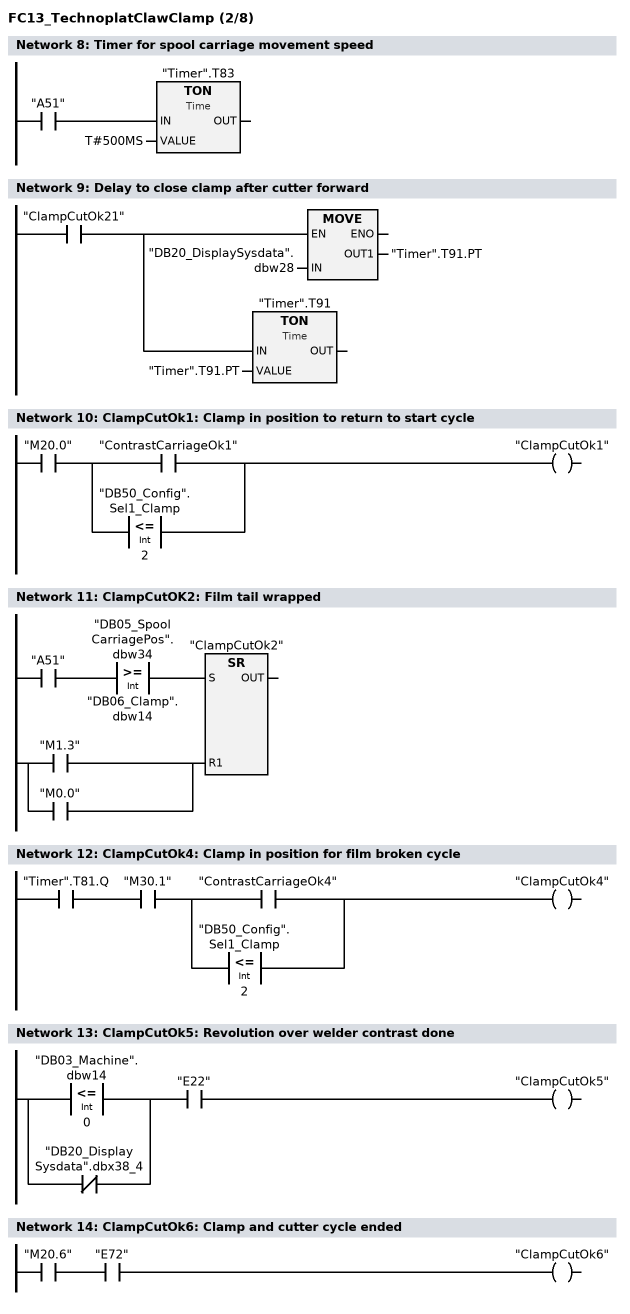
   "Timer".T83.TON(IN := "A51", PT := T#500MS);   // TON coil
END_REGION

REGION Network 9: Delay to close clamp after cutter forward
   IF "ClampCutOk21" THEN "Timer".T91.PT := "DB20_DisplaySysdata".dbw28; END_IF;
   "Timer".T91.TON(IN := "ClampCutOk21", PT := "Timer".T91.PT);   // TON coil
END_REGION

REGION Network 10: ClampCutOk1: Clamp in position to return to start cycle
   RUNG wire#powerrail
      Contact( "M20.0" )
      wire#w1
      Contact( "ContrastCarriageOk1" )
      wire#w2
      Coil( "ClampCutOk1" )
   END_RUNG
   RUNG wire#w1
      { S7_Templates := "SrcType := Int" } LE_Contact(in1 := "DB50_Config".Sel1_Clamp, in2 := 2)
   END_RUNG wire#w2
   // the same network as SCL:
   "ClampCutOk1" := "M20.0" AND ("ContrastCarriageOk1" OR ("DB50_Config".Sel1_Clamp <= 2));
END_REGION

REGION Network 11: ClampCutOK2: Film tail wrapped
   RUNG wire#powerrail
      Contact( "A51" )
      { S7_Templates := "SrcType := Int" } GE_Contact(in1 := "DB05_SpoolCarriagePos".dbw34, in2 := "DB06_Clamp".dbw14)
      S_SR(operand := "ClampCutOk2", r1 := wire#w1)
   END_RUNG
   RUNG wire#powerrail
      Contact( "M1.3" )
   END_RUNG wire#w1
   RUNG wire#powerrail
      Contact( "M0.0" )
   END_RUNG wire#w1
   // the same network as SCL:
   IF "A51" AND ("DB05_SpoolCarriagePos".dbw34 >= "DB06_Clamp".dbw14) THEN
       "ClampCutOk2" := TRUE;   // SR flip-flop
   END_IF;
   IF "M1.3" OR "M0.0" THEN "ClampCutOk2" := FALSE; END_IF;
END_REGION

REGION Network 12: ClampCutOk4: Clamp in position for film broken cycle
   RUNG wire#powerrail
      Contact( "Timer".T81.Q )
      Contact( "M30.1" )
      wire#w1
      Contact( "ContrastCarriageOk4" )
      wire#w2
      Coil( "ClampCutOk4" )
   END_RUNG
   RUNG wire#w1
      { S7_Templates := "SrcType := Int" } LE_Contact(in1 := "DB50_Config".Sel1_Clamp, in2 := 2)
   END_RUNG wire#w2
   // the same network as SCL:
   "ClampCutOk4" := "Timer".T81.Q AND "M30.1" AND ("ContrastCarriageOk4" OR ("DB50_Config".Sel1_Clamp <= 2));
END_REGION

REGION Network 13: ClampCutOk5: Revolution over welder contrast done
   RUNG wire#powerrail
      { S7_Templates := "SrcType := Int" } LE_Contact(in1 := "DB03_Machine".dbw14, in2 := 0)
      wire#w1
      Contact( "E22" )
      Coil( "ClampCutOk5" )
   END_RUNG
   RUNG wire#powerrail
      I_Contact( "DB20_DisplaySysdata".dbx38_4 )
   END_RUNG wire#w1
   // the same network as SCL:
   "ClampCutOk5" := (("DB03_Machine".dbw14 <= 0) OR NOT "DB20_DisplaySysdata".dbx38_4) AND "E22";
END_REGION

REGION Network 14: ClampCutOk6: Clamp and cutter cycle ended
   RUNG wire#powerrail
      Contact( "M20.6" )
      Contact( "E72" )
      Coil( "ClampCutOk6" )
   END_RUNG
   // the same network as SCL:
   "ClampCutOk6" := "M20.6" AND "E72";
END_REGION

REGION Network 15: ClampCutOk7: Clamp and cutter units in position to begin cycle
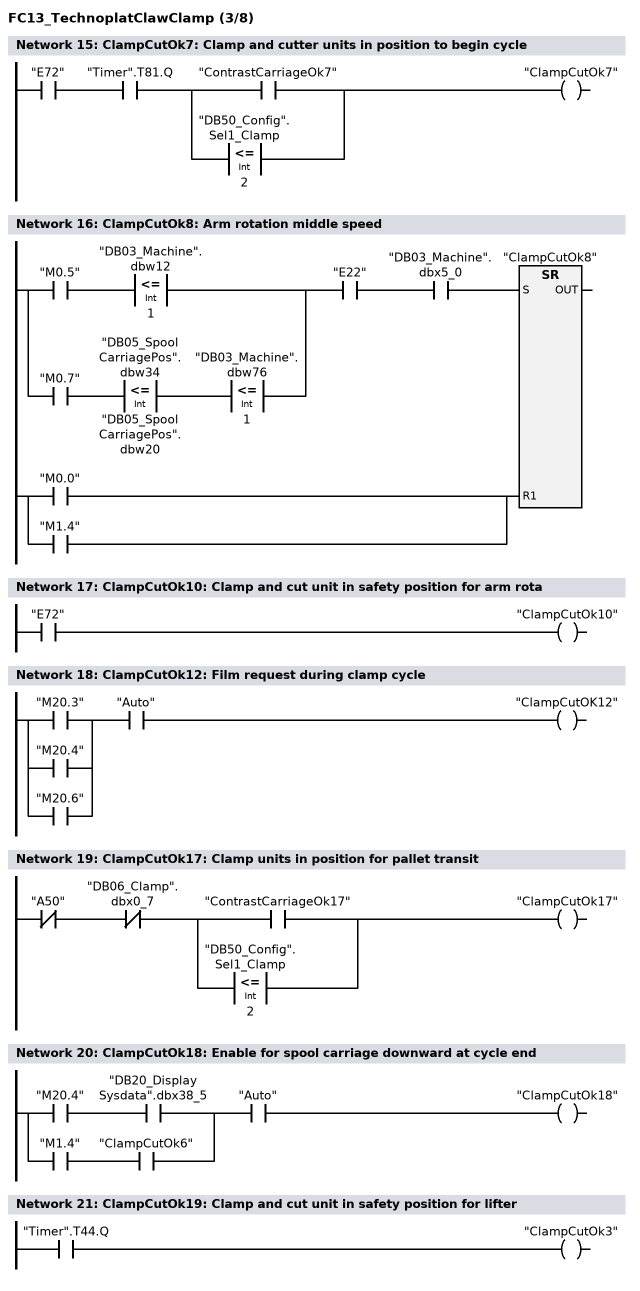
   RUNG wire#powerrail
      Contact( "E72" )
      Contact( "Timer".T81.Q )
      wire#w1
      Contact( "ContrastCarriageOk7" )
      wire#w2
      Coil( "ClampCutOk7" )
   END_RUNG
   RUNG wire#w1
      { S7_Templates := "SrcType := Int" } LE_Contact(in1 := "DB50_Config".Sel1_Clamp, in2 := 2)
   END_RUNG wire#w2
   // the same network as SCL:
   "ClampCutOk7" := "E72" AND "Timer".T81.Q AND ("ContrastCarriageOk7" OR ("DB50_Config".Sel1_Clamp <= 2));
END_REGION

REGION Network 16: ClampCutOk8: Arm rotation middle speed
   RUNG wire#powerrail
      Contact( "M0.5" )
      { S7_Templates := "SrcType := Int" } LE_Contact(in1 := "DB03_Machine".dbw12, in2 := 1)
      wire#w1
      Contact( "E22" )
      Contact( "DB03_Machine".dbx5_0 )
      S_SR(operand := "ClampCutOk8", r1 := wire#w2)
   END_RUNG
   RUNG wire#powerrail
      Contact( "M0.7" )
      { S7_Templates := "SrcType := Int" } LE_Contact(in1 := "DB05_SpoolCarriagePos".dbw34, in2 := "DB05_SpoolCarriagePos".dbw20)
      { S7_Templates := "SrcType := Int" } LE_Contact(in1 := "DB03_Machine".dbw76, in2 := 1)
   END_RUNG wire#w1
   RUNG wire#powerrail
      Contact( "M0.0" )
   END_RUNG wire#w2
   RUNG wire#powerrail
      Contact( "M1.4" )
   END_RUNG wire#w2
   // the same network as SCL:
   IF (("M0.5" AND ("DB03_Machine".dbw12 <= 1)) OR ("M0.7" AND ("DB05_SpoolCarriagePos".dbw34 <= "DB05_SpoolCarriagePos".dbw20) AND ("DB03_Machine".dbw76 <= 1))) AND "E22" AND "DB03_Machine".dbx5_0 THEN
       "ClampCutOk8" := TRUE;   // SR flip-flop
   END_IF;
   IF "M0.0" OR "M1.4" THEN "ClampCutOk8" := FALSE; END_IF;
END_REGION

REGION Network 17: ClampCutOk10: Clamp and cut unit in safety position for arm rota
   RUNG wire#powerrail
      Contact( "E72" )
      Coil( "ClampCutOk10" )
   END_RUNG
   // the same network as SCL:
   "ClampCutOk10" := "E72";
END_REGION

REGION Network 18: ClampCutOk12: Film request during clamp cycle
   RUNG wire#powerrail
      Contact( "M20.3" )
      wire#w1
      Contact( "Auto" )
      Coil( "ClampCutOK12" )
   END_RUNG
   RUNG wire#powerrail
      Contact( "M20.4" )
   END_RUNG wire#w1
   RUNG wire#powerrail
      Contact( "M20.6" )
   END_RUNG wire#w1
   // the same network as SCL:
   "ClampCutOK12" := ("M20.3" OR "M20.4" OR "M20.6") AND "Auto";
END_REGION

REGION Network 19: ClampCutOk17: Clamp units in position for pallet transit
   RUNG wire#powerrail
      I_Contact( "A50" )
      I_Contact( "DB06_Clamp".dbx0_7 )
      wire#w1
      Contact( "ContrastCarriageOk17" )
      wire#w2
      Coil( "ClampCutOk17" )
   END_RUNG
   RUNG wire#w1
      { S7_Templates := "SrcType := Int" } LE_Contact(in1 := "DB50_Config".Sel1_Clamp, in2 := 2)
   END_RUNG wire#w2
   // the same network as SCL:
   "ClampCutOk17" := NOT "A50" AND NOT "DB06_Clamp".dbx0_7 AND ("ContrastCarriageOk17" OR ("DB50_Config".Sel1_Clamp <= 2));
END_REGION

REGION Network 20: ClampCutOk18: Enable for spool carriage downward at cycle end
   RUNG wire#powerrail
      Contact( "M20.4" )
      Contact( "DB20_DisplaySysdata".dbx38_5 )
      wire#w1
      Contact( "Auto" )
      Coil( "ClampCutOk18" )
   END_RUNG
   RUNG wire#powerrail
      Contact( "M1.4" )
      Contact( "ClampCutOk6" )
   END_RUNG wire#w1
   // the same network as SCL:
   "ClampCutOk18" := (("M20.4" AND "DB20_DisplaySysdata".dbx38_5) OR ("M1.4" AND "ClampCutOk6")) AND "Auto";
END_REGION

REGION Network 21: ClampCutOk19: Clamp and cut unit in safety position for lifter
   RUNG wire#powerrail
      Contact( "Timer".T44.Q )
      Coil( "ClampCutOk3" )
   END_RUNG
   // the same network as SCL:
   "ClampCutOk3" := "Timer".T44.Q;
END_REGION

REGION Network 22: ClampCutOk11: Exclude deceleration not correct alarm
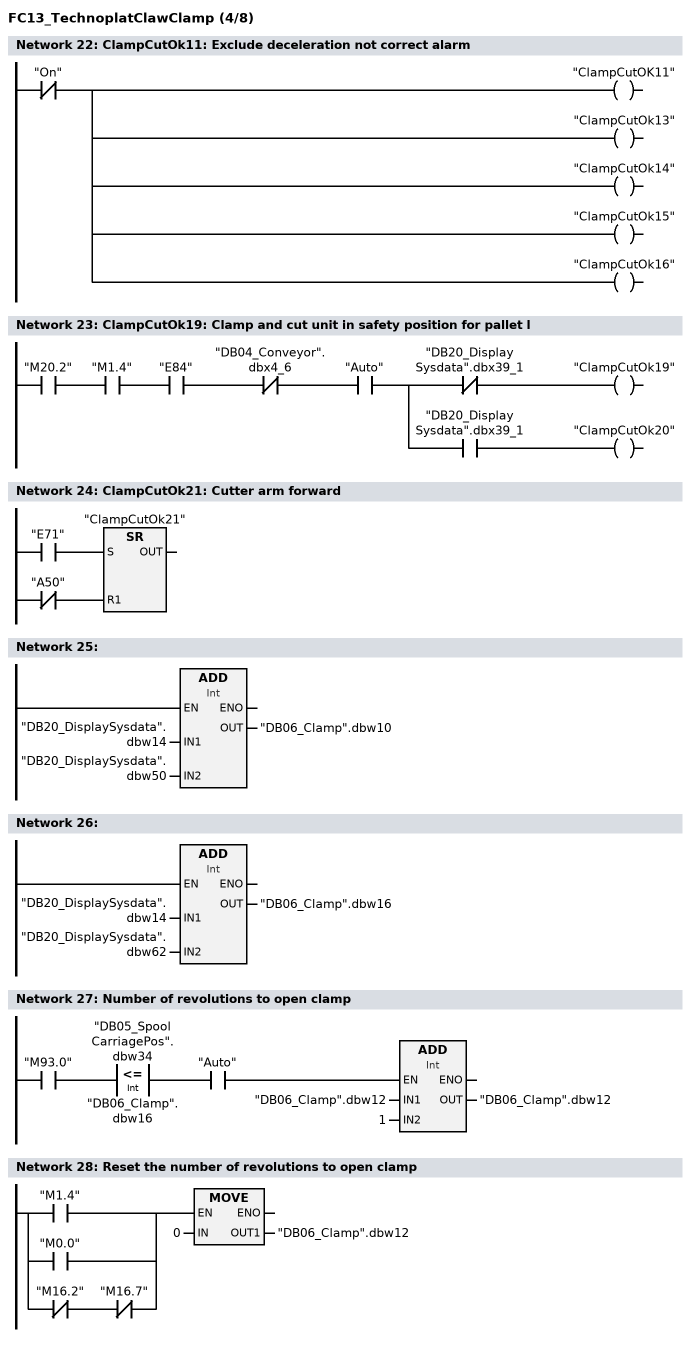
   RUNG wire#powerrail
      I_Contact( "On" )
      wire#w1
      Coil( "ClampCutOK11" )
   END_RUNG
   RUNG wire#w1
      Coil( "ClampCutOk13" )
   END_RUNG
   RUNG wire#w1
      Coil( "ClampCutOk14" )
   END_RUNG
   RUNG wire#w1
      Coil( "ClampCutOk15" )
   END_RUNG
   RUNG wire#w1
      Coil( "ClampCutOk16" )
   END_RUNG
   // the same network as SCL:
   "ClampCutOK11" := NOT "On";
   "ClampCutOk13" := NOT "On";
   "ClampCutOk14" := NOT "On";
   "ClampCutOk15" := NOT "On";
   "ClampCutOk16" := NOT "On";
END_REGION

REGION Network 23: ClampCutOk19: Clamp and cut unit in safety position for pallet l
   RUNG wire#powerrail
      Contact( "M20.2" )
      Contact( "M1.4" )
      Contact( "E84" )
      I_Contact( "DB04_Conveyor".dbx4_6 )
      Contact( "Auto" )
      wire#w1
      I_Contact( "DB20_DisplaySysdata".dbx39_1 )
      Coil( "ClampCutOk19" )
   END_RUNG
   RUNG wire#w1
      Contact( "DB20_DisplaySysdata".dbx39_1 )
      Coil( "ClampCutOk20" )
   END_RUNG
   // the same network as SCL:
   #_w1 := "M20.2" AND "M1.4" AND "E84" AND NOT "DB04_Conveyor".dbx4_6 AND "Auto";
   "ClampCutOk19" := #_w1 AND NOT "DB20_DisplaySysdata".dbx39_1;
   "ClampCutOk20" := #_w1 AND "DB20_DisplaySysdata".dbx39_1;
END_REGION

REGION Network 24: ClampCutOk21: Cutter arm forward
   RUNG wire#powerrail
      Contact( "E71" )
      S_SR(operand := "ClampCutOk21", r1 := wire#w1)
   END_RUNG
   RUNG wire#powerrail
      I_Contact( "A50" )
   END_RUNG wire#w1
   // the same network as SCL:
   IF "E71" THEN
       "ClampCutOk21" := TRUE;   // SR flip-flop
   END_IF;
   IF NOT "A50" THEN "ClampCutOk21" := FALSE; END_IF;
END_REGION

REGION Network 25
   RUNG wire#powerrail
      { S7_Templates := "SrcType := Int"; S7_GenerateENO := "TRUE" } Add(in1 := "DB20_DisplaySysdata".dbw14, in2 := "DB20_DisplaySysdata".dbw50, out => "DB06_Clamp".dbw10)
   END_RUNG
   // the same network as SCL:
   "DB06_Clamp".dbw10 := "DB20_DisplaySysdata".dbw14 + "DB20_DisplaySysdata".dbw50;
END_REGION

REGION Network 26
   RUNG wire#powerrail
      { S7_Templates := "SrcType := Int"; S7_GenerateENO := "TRUE" } Add(in1 := "DB20_DisplaySysdata".dbw14, in2 := "DB20_DisplaySysdata".dbw62, out => "DB06_Clamp".dbw16)
   END_RUNG
   // the same network as SCL:
   "DB06_Clamp".dbw16 := "DB20_DisplaySysdata".dbw14 + "DB20_DisplaySysdata".dbw62;
END_REGION

REGION Network 27: Number of revolutions to open clamp
   RUNG wire#powerrail
      Contact( "M93.0" )
      { S7_Templates := "SrcType := Int" } LE_Contact(in1 := "DB05_SpoolCarriagePos".dbw34, in2 := "DB06_Clamp".dbw16)
      Contact( "Auto" )
      { S7_Templates := "SrcType := Int"; S7_GenerateENO := "TRUE" } Add(in1 := "DB06_Clamp".dbw12, in2 := 1, out => "DB06_Clamp".dbw12)
   END_RUNG
   // the same network as SCL:
   IF "M93.0" AND ("DB05_SpoolCarriagePos".dbw34 <= "DB06_Clamp".dbw16) AND "Auto" THEN
       "DB06_Clamp".dbw12 := "DB06_Clamp".dbw12 + 1;
   END_IF;
END_REGION

REGION Network 28: Reset the number of revolutions to open clamp
   RUNG wire#powerrail
      Contact( "M1.4" )
      wire#w1
      { S7_GenerateENO := "TRUE" } Move(in := 0, out1 => "DB06_Clamp".dbw12)
   END_RUNG
   RUNG wire#powerrail
      Contact( "M0.0" )
   END_RUNG wire#w1
   RUNG wire#powerrail
      I_Contact( "M16.2" )
      I_Contact( "M16.7" )
   END_RUNG wire#w1
   // the same network as SCL:
   IF "M1.4" OR "M0.0" OR (NOT "M16.2" AND NOT "M16.7") THEN "DB06_Clamp".dbw12 := 0; END_IF;
END_REGION

REGION Network 29
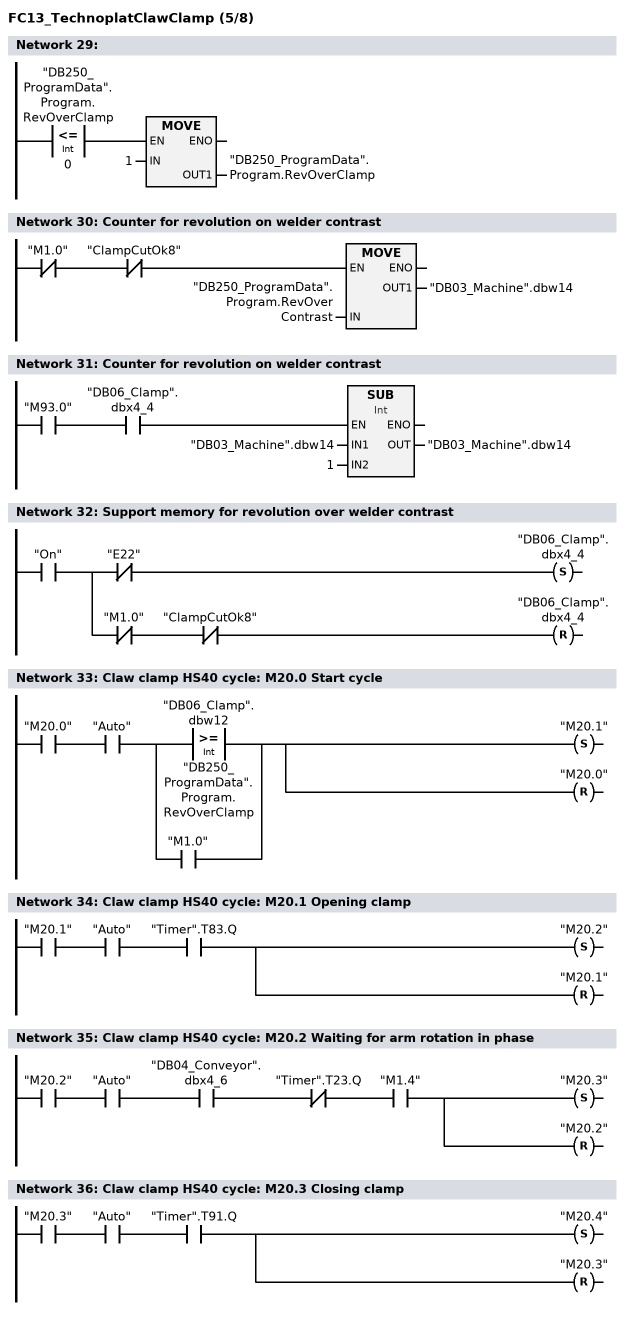
   RUNG wire#powerrail
      { S7_Templates := "SrcType := Int" } LE_Contact(in1 := "DB250_ProgramData".Program.RevOverClamp, in2 := 0)
      { S7_GenerateENO := "TRUE" } Move(in := 1, out1 => "DB250_ProgramData".Program.RevOverClamp)
   END_RUNG
   // the same network as SCL:
   IF "DB250_ProgramData".Program.RevOverClamp <= 0 THEN
       "DB250_ProgramData".Program.RevOverClamp := 1;
   END_IF;
END_REGION

REGION Network 30: Counter for revolution on welder contrast
   RUNG wire#powerrail
      I_Contact( "M1.0" )
      I_Contact( "ClampCutOk8" )
      { S7_GenerateENO := "TRUE" } Move(in := "DB250_ProgramData".Program.RevOverContrast, out1 => "DB03_Machine".dbw14)
   END_RUNG
   // the same network as SCL:
   IF NOT "M1.0" AND NOT "ClampCutOk8" THEN
       "DB03_Machine".dbw14 := "DB250_ProgramData".Program.RevOverContrast;
   END_IF;
END_REGION

REGION Network 31: Counter for revolution on welder contrast
   RUNG wire#powerrail
      Contact( "M93.0" )
      Contact( "DB06_Clamp".dbx4_4 )
      { S7_Templates := "SrcType := Int"; S7_GenerateENO := "TRUE" } Sub(in1 := "DB03_Machine".dbw14, in2 := 1, out => "DB03_Machine".dbw14)
   END_RUNG
   // the same network as SCL:
   IF "M93.0" AND "DB06_Clamp".dbx4_4 THEN "DB03_Machine".dbw14 := "DB03_Machine".dbw14 - 1; END_IF;
END_REGION

REGION Network 32: Support memory for revolution over welder contrast
   RUNG wire#powerrail
      Contact( "On" )
      wire#w1
      I_Contact( "E22" )
      S_Coil( "DB06_Clamp".dbx4_4 )
   END_RUNG
   RUNG wire#w1
      I_Contact( "M1.0" )
      I_Contact( "ClampCutOk8" )
      R_Coil( "DB06_Clamp".dbx4_4 )
   END_RUNG
   // the same network as SCL:
   IF "On" AND NOT "E22" THEN "DB06_Clamp".dbx4_4 := TRUE; END_IF;
   IF "On" AND NOT "M1.0" AND NOT "ClampCutOk8" THEN "DB06_Clamp".dbx4_4 := FALSE; END_IF;
END_REGION

REGION Network 33: Claw clamp HS40 cycle: M20.0 Start cycle
   RUNG wire#powerrail
      Contact( "M20.0" )
      Contact( "Auto" )
      wire#w1
      { S7_Templates := "SrcType := Int" } GE_Contact(in1 := "DB06_Clamp".dbw12, in2 := "DB250_ProgramData".Program.RevOverClamp)
      wire#w2
      S_Coil( "M20.1" )
   END_RUNG
   RUNG wire#w1
      Contact( "M1.0" )
   END_RUNG wire#w2
   RUNG wire#w2
      R_Coil( "M20.0" )
   END_RUNG
   // the same network as SCL:
   IF "M20.0" AND "Auto" AND (("DB06_Clamp".dbw12 >= "DB250_ProgramData".Program.RevOverClamp) OR "M1.0") THEN
       "M20.1" := TRUE;
       "M20.0" := FALSE;
   END_IF;
END_REGION

REGION Network 34: Claw clamp HS40 cycle: M20.1 Opening clamp
   RUNG wire#powerrail
      Contact( "M20.1" )
      Contact( "Auto" )
      Contact( "Timer".T83.Q )
      wire#w1
      S_Coil( "M20.2" )
   END_RUNG
   RUNG wire#w1
      R_Coil( "M20.1" )
   END_RUNG
   // the same network as SCL:
   IF "M20.1" AND "Auto" AND "Timer".T83.Q THEN
       "M20.2" := TRUE;
       "M20.1" := FALSE;
   END_IF;
END_REGION

REGION Network 35: Claw clamp HS40 cycle: M20.2 Waiting for arm rotation in phase
   RUNG wire#powerrail
      Contact( "M20.2" )
      Contact( "Auto" )
      Contact( "DB04_Conveyor".dbx4_6 )
      I_Contact( "Timer".T23.Q )
      Contact( "M1.4" )
      wire#w1
      S_Coil( "M20.3" )
   END_RUNG
   RUNG wire#w1
      R_Coil( "M20.2" )
   END_RUNG
   // the same network as SCL:
   IF "M20.2" AND "Auto" AND "DB04_Conveyor".dbx4_6 AND NOT "Timer".T23.Q AND "M1.4" THEN
       "M20.3" := TRUE;
       "M20.2" := FALSE;
   END_IF;
END_REGION

REGION Network 36: Claw clamp HS40 cycle: M20.3 Closing clamp
   RUNG wire#powerrail
      Contact( "M20.3" )
      Contact( "Auto" )
      Contact( "Timer".T91.Q )
      wire#w1
      S_Coil( "M20.4" )
   END_RUNG
   RUNG wire#w1
      R_Coil( "M20.3" )
   END_RUNG
   // the same network as SCL:
   IF "M20.3" AND "Auto" AND "Timer".T91.Q THEN
       "M20.4" := TRUE;
       "M20.3" := FALSE;
   END_IF;
END_REGION

REGION Network 37: Claw clamp HS40 cycle: M20.4 Welder and cut unit forward
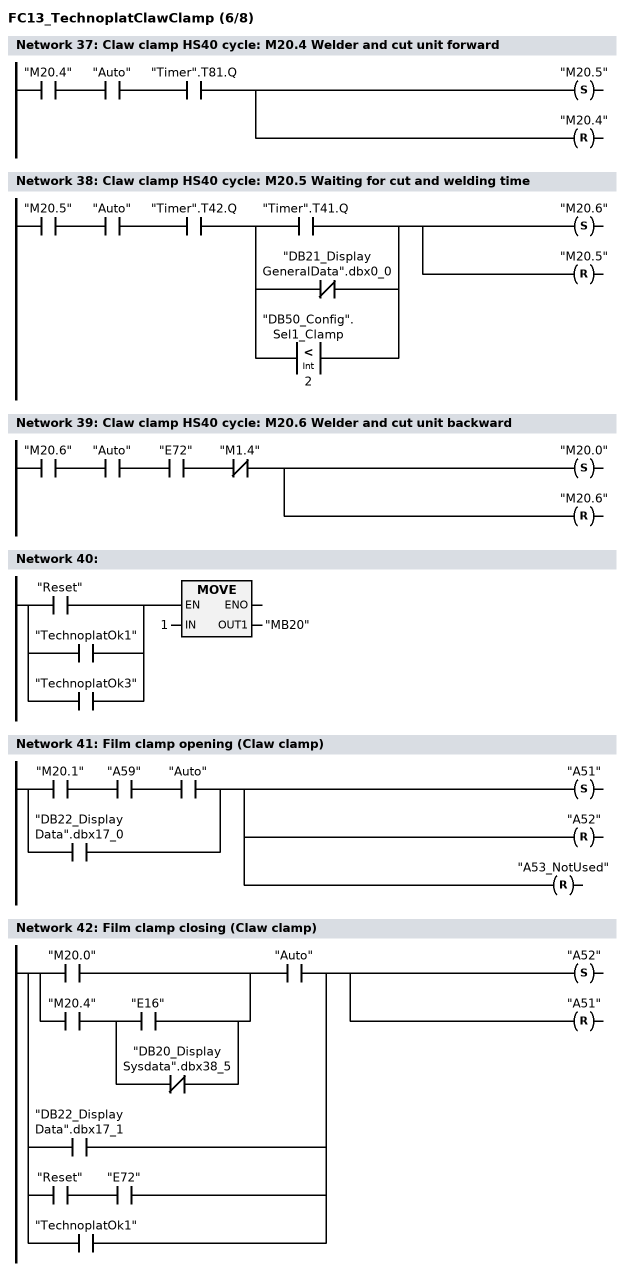
   RUNG wire#powerrail
      Contact( "M20.4" )
      Contact( "Auto" )
      Contact( "Timer".T81.Q )
      wire#w1
      S_Coil( "M20.5" )
   END_RUNG
   RUNG wire#w1
      R_Coil( "M20.4" )
   END_RUNG
   // the same network as SCL:
   IF "M20.4" AND "Auto" AND "Timer".T81.Q THEN
       "M20.5" := TRUE;
       "M20.4" := FALSE;
   END_IF;
END_REGION

REGION Network 38: Claw clamp HS40 cycle: M20.5 Waiting for cut and welding time
   RUNG wire#powerrail
      Contact( "M20.5" )
      Contact( "Auto" )
      Contact( "Timer".T42.Q )
      wire#w1
      Contact( "Timer".T41.Q )
      wire#w2
      S_Coil( "M20.6" )
   END_RUNG
   RUNG wire#w1
      I_Contact( "DB21_DisplayGeneralData".dbx0_0 )
   END_RUNG wire#w2
   RUNG wire#w1
      { S7_Templates := "SrcType := Int" } LT_Contact(in1 := "DB50_Config".Sel1_Clamp, in2 := 2)
   END_RUNG wire#w2
   RUNG wire#w2
      R_Coil( "M20.5" )
   END_RUNG
   // the same network as SCL:
   IF "M20.5" AND "Auto" AND "Timer".T42.Q AND ("Timer".T41.Q OR NOT "DB21_DisplayGeneralData".dbx0_0 OR ("DB50_Config".Sel1_Clamp < 2)) THEN
       "M20.6" := TRUE;
       "M20.5" := FALSE;
   END_IF;
END_REGION

REGION Network 39: Claw clamp HS40 cycle: M20.6 Welder and cut unit backward
   RUNG wire#powerrail
      Contact( "M20.6" )
      Contact( "Auto" )
      Contact( "E72" )
      I_Contact( "M1.4" )
      wire#w1
      S_Coil( "M20.0" )
   END_RUNG
   RUNG wire#w1
      R_Coil( "M20.6" )
   END_RUNG
   // the same network as SCL:
   IF "M20.6" AND "Auto" AND "E72" AND NOT "M1.4" THEN
       "M20.0" := TRUE;
       "M20.6" := FALSE;
   END_IF;
END_REGION

REGION Network 40
   RUNG wire#powerrail
      Contact( "Reset" )
      wire#w1
      { S7_GenerateENO := "TRUE" } Move(in := 1, out1 => "MB20")
   END_RUNG
   RUNG wire#powerrail
      Contact( "TechnoplatOk1" )
   END_RUNG wire#w1
   RUNG wire#powerrail
      Contact( "TechnoplatOk3" )
   END_RUNG wire#w1
   // the same network as SCL:
   IF "Reset" OR "TechnoplatOk1" OR "TechnoplatOk3" THEN "MB20" := 1; END_IF;
END_REGION

REGION Network 41: Film clamp opening (Claw clamp)
   RUNG wire#powerrail
      Contact( "M20.1" )
      Contact( "A59" )
      Contact( "Auto" )
      wire#w1
      S_Coil( "A51" )
   END_RUNG
   RUNG wire#powerrail
      Contact( "DB22_DisplayData".dbx17_0 )
   END_RUNG wire#w1
   RUNG wire#w1
      R_Coil( "A52" )
   END_RUNG
   RUNG wire#w1
      R_Coil( "A53_NotUsed" )
   END_RUNG
   // the same network as SCL:
   IF ("M20.1" AND "A59" AND "Auto") OR "DB22_DisplayData".dbx17_0 THEN
       "A51" := TRUE;
       "A52" := FALSE;
       "A53_NotUsed" := FALSE;
   END_IF;
END_REGION

REGION Network 42: Film clamp closing (Claw clamp)
   RUNG wire#powerrail
      Contact( "M20.0" )
      wire#w1
      Contact( "Auto" )
      wire#w3
      S_Coil( "A52" )
   END_RUNG
   RUNG wire#powerrail
      Contact( "M20.4" )
      wire#w2
      Contact( "E16" )
   END_RUNG wire#w1
   RUNG wire#w2
      I_Contact( "DB20_DisplaySysdata".dbx38_5 )
   END_RUNG wire#w1
   RUNG wire#powerrail
      Contact( "DB22_DisplayData".dbx17_1 )
   END_RUNG wire#w3
   RUNG wire#powerrail
      Contact( "Reset" )
      Contact( "E72" )
   END_RUNG wire#w3
   RUNG wire#powerrail
      Contact( "TechnoplatOk1" )
   END_RUNG wire#w3
   RUNG wire#w3
      R_Coil( "A51" )
   END_RUNG
   // the same network as SCL:
   IF (("M20.0" OR ("M20.4" AND ("E16" OR NOT "DB20_DisplaySysdata".dbx38_5))) AND "Auto") OR "DB22_DisplayData".dbx17_1 OR ("Reset" AND "E72") OR "TechnoplatOk1" THEN
       "A52" := TRUE;
       "A51" := FALSE;
   END_IF;
END_REGION

REGION Network 43: Film clamp double closing (Claw clamp)
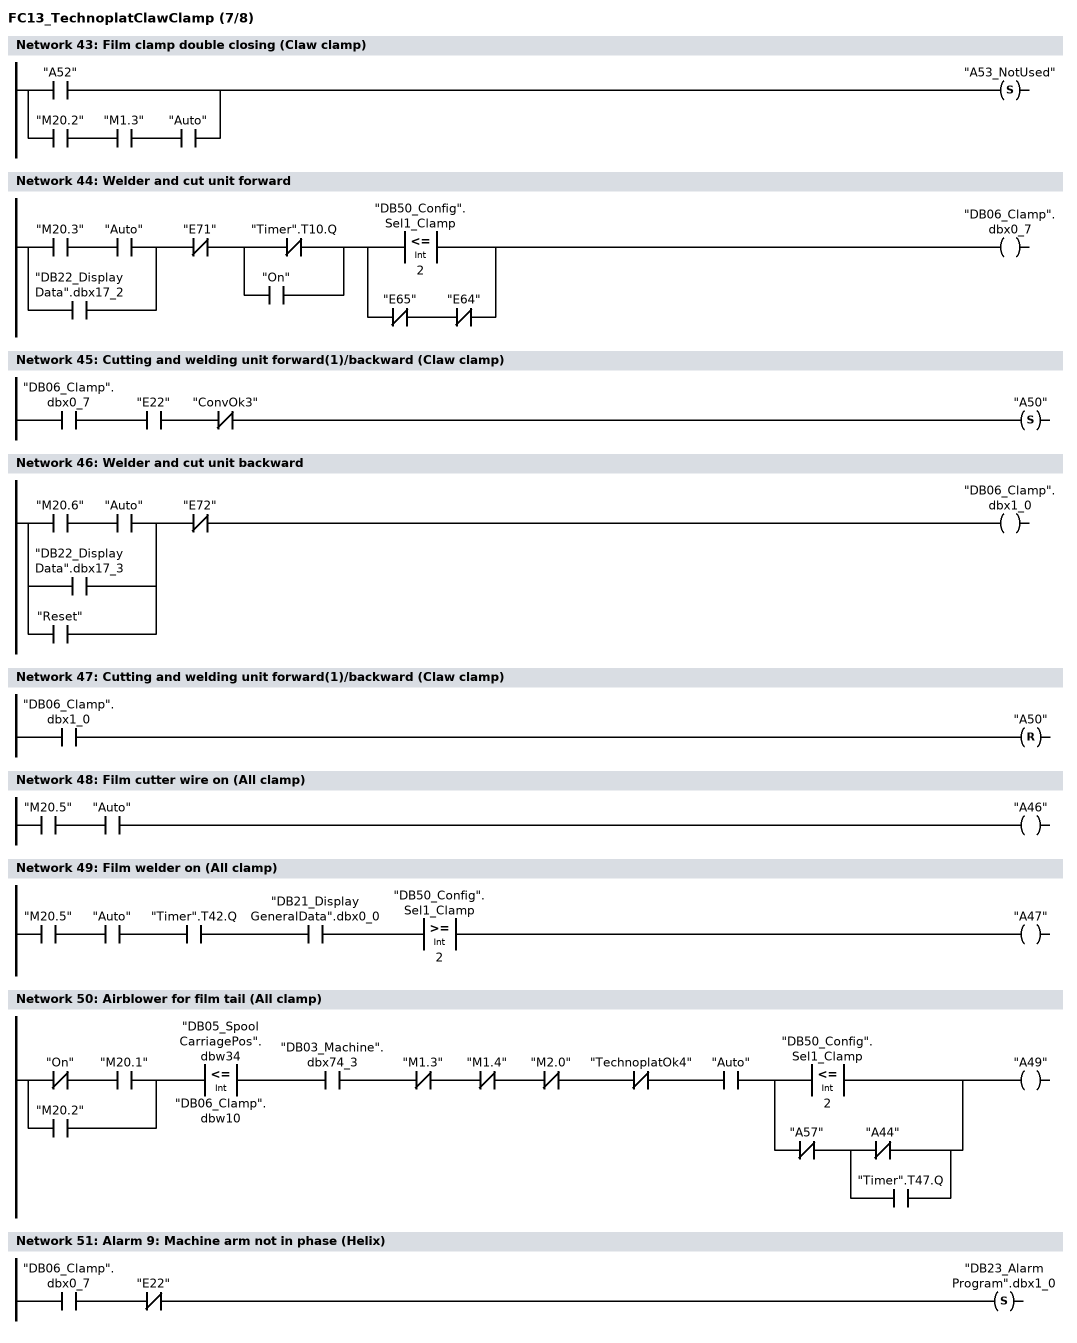
   RUNG wire#powerrail
      Contact( "A52" )
      wire#w1
      S_Coil( "A53_NotUsed" )
   END_RUNG
   RUNG wire#powerrail
      Contact( "M20.2" )
      Contact( "M1.3" )
      Contact( "Auto" )
   END_RUNG wire#w1
   // the same network as SCL:
   IF "A52" OR ("M20.2" AND "M1.3" AND "Auto") THEN "A53_NotUsed" := TRUE; END_IF;
END_REGION

REGION Network 44: Welder and cut unit forward
   RUNG wire#powerrail
      Contact( "M20.3" )
      Contact( "Auto" )
      wire#w1
      I_Contact( "E71" )
      wire#w2
      I_Contact( "Timer".T10.Q )
      wire#w3
      { S7_Templates := "SrcType := Int" } LE_Contact(in1 := "DB50_Config".Sel1_Clamp, in2 := 2)
      wire#w4
      Coil( "DB06_Clamp".dbx0_7 )
   END_RUNG
   RUNG wire#powerrail
      Contact( "DB22_DisplayData".dbx17_2 )
   END_RUNG wire#w1
   RUNG wire#w2
      Contact( "On" )
   END_RUNG wire#w3
   RUNG wire#w3
      I_Contact( "E65" )
      I_Contact( "E64" )
   END_RUNG wire#w4
   // the same network as SCL:
   "DB06_Clamp".dbx0_7 := (("M20.3" AND "Auto") OR "DB22_DisplayData".dbx17_2) AND NOT "E71" AND (NOT "Timer".T10.Q OR "On") AND (("DB50_Config".Sel1_Clamp <= 2) OR (NOT "E65" AND NOT "E64"));
END_REGION

REGION Network 45: Cutting and welding unit forward(1)/backward (Claw clamp)
   RUNG wire#powerrail
      Contact( "DB06_Clamp".dbx0_7 )
      Contact( "E22" )
      I_Contact( "ConvOk3" )
      S_Coil( "A50" )
   END_RUNG
   // the same network as SCL:
   IF "DB06_Clamp".dbx0_7 AND "E22" AND NOT "ConvOk3" THEN "A50" := TRUE; END_IF;
END_REGION

REGION Network 46: Welder and cut unit backward
   RUNG wire#powerrail
      Contact( "M20.6" )
      Contact( "Auto" )
      wire#w1
      I_Contact( "E72" )
      Coil( "DB06_Clamp".dbx1_0 )
   END_RUNG
   RUNG wire#powerrail
      Contact( "DB22_DisplayData".dbx17_3 )
   END_RUNG wire#w1
   RUNG wire#powerrail
      Contact( "Reset" )
   END_RUNG wire#w1
   // the same network as SCL:
   "DB06_Clamp".dbx1_0 := (("M20.6" AND "Auto") OR "DB22_DisplayData".dbx17_3 OR "Reset") AND NOT "E72";
END_REGION

REGION Network 47: Cutting and welding unit forward(1)/backward (Claw clamp)
   RUNG wire#powerrail
      Contact( "DB06_Clamp".dbx1_0 )
      R_Coil( "A50" )
   END_RUNG
   // the same network as SCL:
   IF "DB06_Clamp".dbx1_0 THEN "A50" := FALSE; END_IF;
END_REGION

REGION Network 48: Film cutter wire on (All clamp)
   RUNG wire#powerrail
      Contact( "M20.5" )
      Contact( "Auto" )
      Coil( "A46" )
   END_RUNG
   // the same network as SCL:
   "A46" := "M20.5" AND "Auto";
END_REGION

REGION Network 49: Film welder on (All clamp)
   RUNG wire#powerrail
      Contact( "M20.5" )
      Contact( "Auto" )
      Contact( "Timer".T42.Q )
      Contact( "DB21_DisplayGeneralData".dbx0_0 )
      { S7_Templates := "SrcType := Int" } GE_Contact(in1 := "DB50_Config".Sel1_Clamp, in2 := 2)
      Coil( "A47" )
   END_RUNG
   // the same network as SCL:
   "A47" := "M20.5" AND "Auto" AND "Timer".T42.Q AND "DB21_DisplayGeneralData".dbx0_0 AND ("DB50_Config".Sel1_Clamp >= 2);
END_REGION

REGION Network 50: Airblower for film tail (All clamp)
   RUNG wire#powerrail
      I_Contact( "On" )
      Contact( "M20.1" )
      wire#w1
      { S7_Templates := "SrcType := Int" } LE_Contact(in1 := "DB05_SpoolCarriagePos".dbw34, in2 := "DB06_Clamp".dbw10)
      Contact( "DB03_Machine".dbx74_3 )
      I_Contact( "M1.3" )
      I_Contact( "M1.4" )
      I_Contact( "M2.0" )
      I_Contact( "TechnoplatOk4" )
      Contact( "Auto" )
      wire#w2
      { S7_Templates := "SrcType := Int" } LE_Contact(in1 := "DB50_Config".Sel1_Clamp, in2 := 2)
      wire#w3
      Coil( "A49" )
   END_RUNG
   RUNG wire#powerrail
      Contact( "M20.2" )
   END_RUNG wire#w1
   RUNG wire#w2
      I_Contact( "A57" )
      wire#w4
      I_Contact( "A44" )
   END_RUNG wire#w3
   RUNG wire#w4
      Contact( "Timer".T47.Q )
   END_RUNG wire#w3
   // the same network as SCL:
   "A49" := ((NOT "On" AND "M20.1") OR "M20.2") AND ("DB05_SpoolCarriagePos".dbw34 <= "DB06_Clamp".dbw10) AND "DB03_Machine".dbx74_3 AND NOT "M1.3" AND NOT "M1.4" AND NOT "M2.0" AND NOT "TechnoplatOk4" AND "Auto" AND (("DB50_Config".Sel1_Clamp <= 2) OR (NOT "A57" AND (NOT "A44" OR "Timer".T47.Q)));
END_REGION

REGION Network 51: Alarm 9: Machine arm not in phase (Helix)
   RUNG wire#powerrail
      Contact( "DB06_Clamp".dbx0_7 )
      I_Contact( "E22" )
      S_Coil( "DB23_AlarmProgram".dbx1_0 )
   END_RUNG
   // the same network as SCL:
   IF "DB06_Clamp".dbx0_7 AND NOT "E22" THEN "DB23_AlarmProgram".dbx1_0 := TRUE; END_IF;
END_REGION

REGION Network 52: Alarm 52: Check the welder circuit (Clamp)
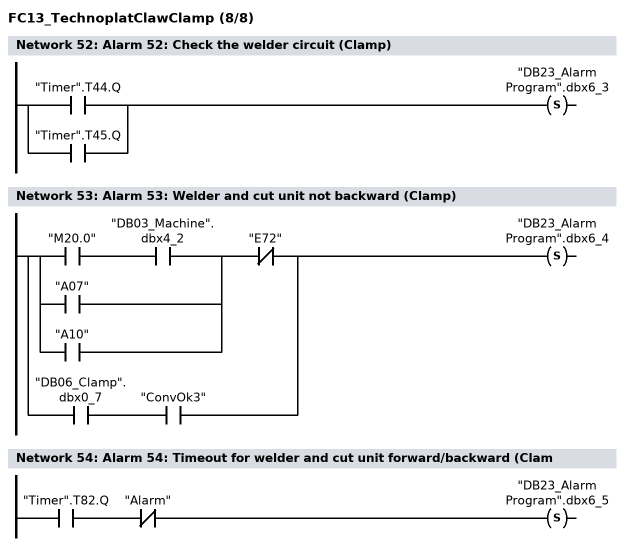
   RUNG wire#powerrail
      Contact( "Timer".T44.Q )
      wire#w1
      S_Coil( "DB23_AlarmProgram".dbx6_3 )
   END_RUNG
   RUNG wire#powerrail
      Contact( "Timer".T45.Q )
   END_RUNG wire#w1
   // the same network as SCL:
   IF "Timer".T44.Q OR "Timer".T45.Q THEN "DB23_AlarmProgram".dbx6_3 := TRUE; END_IF;
END_REGION

REGION Network 53: Alarm 53: Welder and cut unit not backward (Clamp)
   RUNG wire#powerrail
      Contact( "M20.0" )
      Contact( "DB03_Machine".dbx4_2 )
      wire#w1
      I_Contact( "E72" )
      wire#w2
      S_Coil( "DB23_AlarmProgram".dbx6_4 )
   END_RUNG
   RUNG wire#powerrail
      Contact( "A07" )
   END_RUNG wire#w1
   RUNG wire#powerrail
      Contact( "A10" )
   END_RUNG wire#w1
   RUNG wire#powerrail
      Contact( "DB06_Clamp".dbx0_7 )
      Contact( "ConvOk3" )
   END_RUNG wire#w2
   // the same network as SCL:
   IF ((("M20.0" AND "DB03_Machine".dbx4_2) OR "A07" OR "A10") AND NOT "E72") OR ("DB06_Clamp".dbx0_7 AND "ConvOk3") THEN
       "DB23_AlarmProgram".dbx6_4 := TRUE;
   END_IF;
END_REGION

REGION Network 54: Alarm 54: Timeout for welder and cut unit forward/backward (Clam
   RUNG wire#powerrail
      Contact( "Timer".T82.Q )
      I_Contact( "Alarm" )
      S_Coil( "DB23_AlarmProgram".dbx6_5 )
   END_RUNG
   // the same network as SCL:
   IF "Timer".T82.Q AND NOT "Alarm" THEN "DB23_AlarmProgram".dbx6_5 := TRUE; END_IF;
END_REGION
END_FUNCTION

FUNCTION "FC18_ContrastCarriage" : Void   // FC18, LAD
TITLE = ContrastCarriage
{ S7_Optimized_Access := 'FALSE' }
VERSION : 0.1
// stored: AutoNumber false, IsIECCheckEnabled false, SetENOAutomatically false, UDAEnableTagReadback false
   VAR_TEMP   // added for the SCL form of the ladder/FBD networks
      _w1 : Bool;
   END_VAR
BEGIN

REGION Network 1: Timeout for welder contrast downward
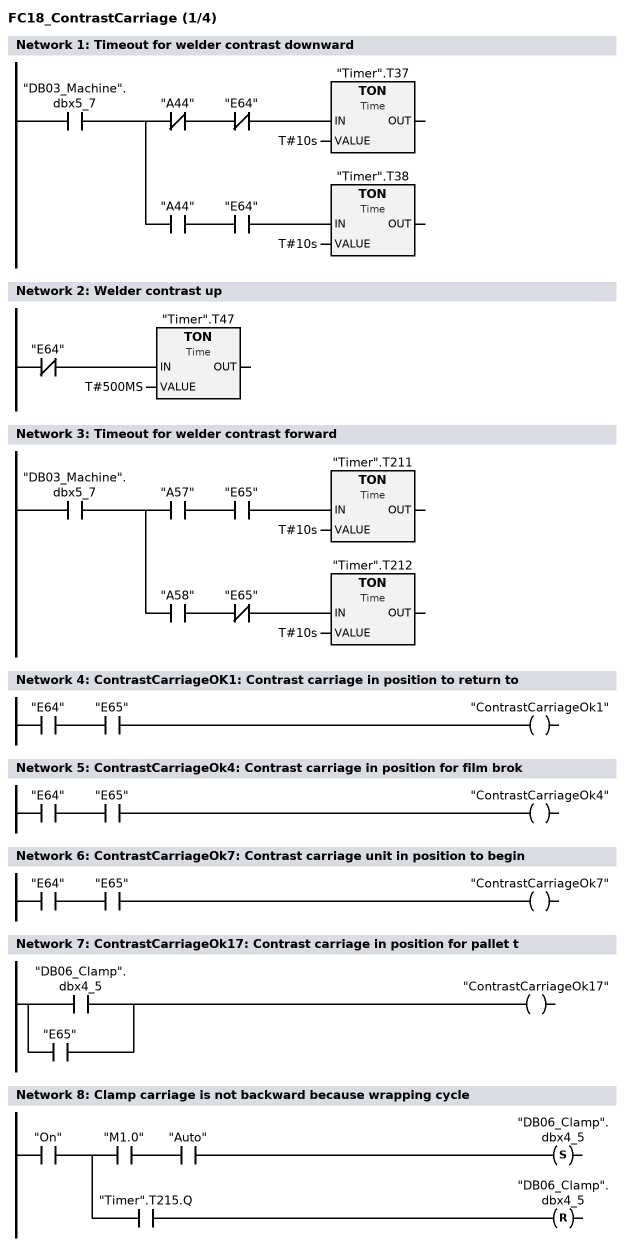
   "Timer".T37.TON(IN := "DB03_Machine".dbx5_7 AND NOT "A44" AND NOT "E64", PT := T#10s);   // TON coil
   "Timer".T38.TON(IN := "DB03_Machine".dbx5_7 AND "A44" AND "E64", PT := T#10s);   // TON coil
END_REGION

REGION Network 2: Welder contrast up
   "Timer".T47.TON(IN := NOT "E64", PT := T#500MS);   // TON coil
END_REGION

REGION Network 3: Timeout for welder contrast forward
   "Timer".T211.TON(IN := "DB03_Machine".dbx5_7 AND "A57" AND "E65", PT := T#10s);   // TON coil
   "Timer".T212.TON(IN := "DB03_Machine".dbx5_7 AND "A58" AND NOT "E65", PT := T#10s);   // TON coil
END_REGION

REGION Network 4: ContrastCarriageOK1: Contrast carriage in position to return to
   RUNG wire#powerrail
      Contact( "E64" )
      Contact( "E65" )
      Coil( "ContrastCarriageOk1" )
   END_RUNG
   // the same network as SCL:
   "ContrastCarriageOk1" := "E64" AND "E65";
END_REGION

REGION Network 5: ContrastCarriageOk4: Contrast carriage in position for film brok
   RUNG wire#powerrail
      Contact( "E64" )
      Contact( "E65" )
      Coil( "ContrastCarriageOk4" )
   END_RUNG
   // the same network as SCL:
   "ContrastCarriageOk4" := "E64" AND "E65";
END_REGION

REGION Network 6: ContrastCarriageOk7: Contrast carriage unit in position to begin
   RUNG wire#powerrail
      Contact( "E64" )
      Contact( "E65" )
      Coil( "ContrastCarriageOk7" )
   END_RUNG
   // the same network as SCL:
   "ContrastCarriageOk7" := "E64" AND "E65";
END_REGION

REGION Network 7: ContrastCarriageOk17: Contrast carriage in position for pallet t
   RUNG wire#powerrail
      Contact( "DB06_Clamp".dbx4_5 )
      wire#w1
      Coil( "ContrastCarriageOk17" )
   END_RUNG
   RUNG wire#powerrail
      Contact( "E65" )
   END_RUNG wire#w1
   // the same network as SCL:
   "ContrastCarriageOk17" := "DB06_Clamp".dbx4_5 OR "E65";
END_REGION

REGION Network 8: Clamp carriage is not backward because wrapping cycle
   RUNG wire#powerrail
      Contact( "On" )
      wire#w1
      Contact( "M1.0" )
      Contact( "Auto" )
      S_Coil( "DB06_Clamp".dbx4_5 )
   END_RUNG
   RUNG wire#w1
      Contact( "Timer".T215.Q )
      R_Coil( "DB06_Clamp".dbx4_5 )
   END_RUNG
   // the same network as SCL:
   IF "On" AND "M1.0" AND "Auto" THEN "DB06_Clamp".dbx4_5 := TRUE; END_IF;
   IF "On" AND "Timer".T215.Q THEN "DB06_Clamp".dbx4_5 := FALSE; END_IF;
END_REGION

REGION Network 9
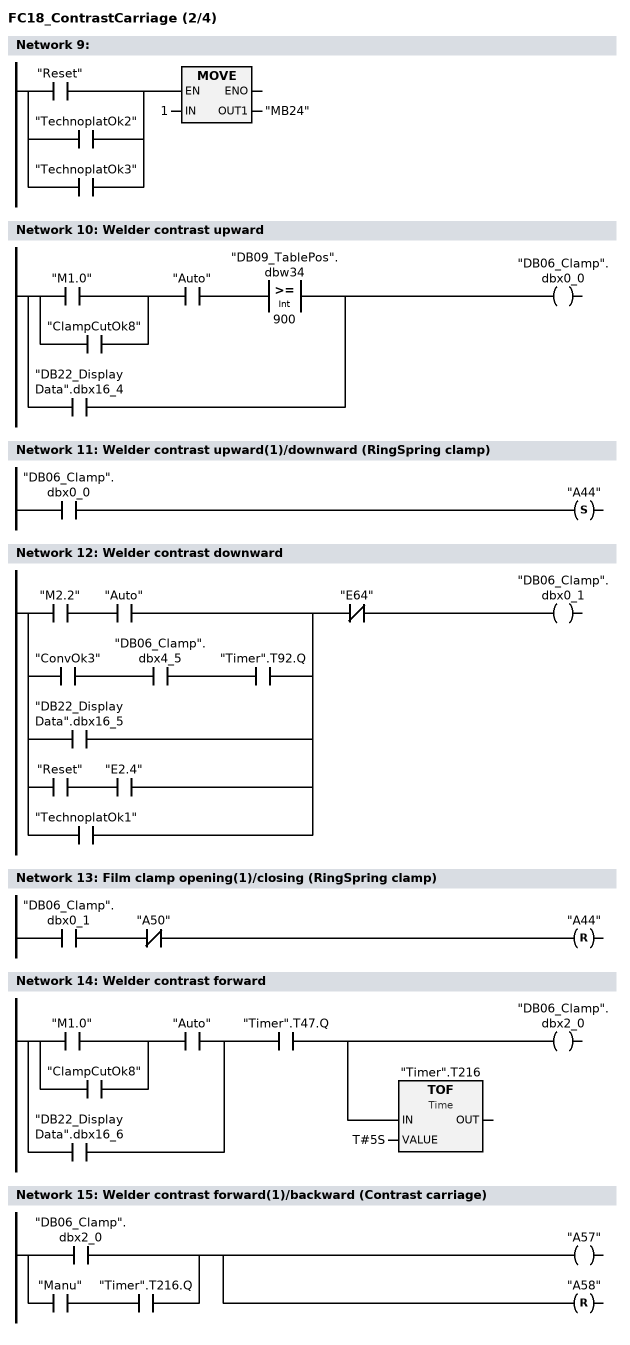
   RUNG wire#powerrail
      Contact( "Reset" )
      wire#w1
      { S7_GenerateENO := "TRUE" } Move(in := 1, out1 => "MB24")
   END_RUNG
   RUNG wire#powerrail
      Contact( "TechnoplatOk2" )
   END_RUNG wire#w1
   RUNG wire#powerrail
      Contact( "TechnoplatOk3" )
   END_RUNG wire#w1
   // the same network as SCL:
   IF "Reset" OR "TechnoplatOk2" OR "TechnoplatOk3" THEN "MB24" := 1; END_IF;
END_REGION

REGION Network 10: Welder contrast upward
   RUNG wire#powerrail
      Contact( "M1.0" )
      wire#w1
      Contact( "Auto" )
      { S7_Templates := "SrcType := Int" } GE_Contact(in1 := "DB09_TablePos".dbw34, in2 := 900)
      wire#w2
      Coil( "DB06_Clamp".dbx0_0 )
   END_RUNG
   RUNG wire#powerrail
      Contact( "ClampCutOk8" )
   END_RUNG wire#w1
   RUNG wire#powerrail
      Contact( "DB22_DisplayData".dbx16_4 )
   END_RUNG wire#w2
   // the same network as SCL:
   "DB06_Clamp".dbx0_0 := (("M1.0" OR "ClampCutOk8") AND "Auto" AND ("DB09_TablePos".dbw34 >= 900)) OR "DB22_DisplayData".dbx16_4;
END_REGION

REGION Network 11: Welder contrast upward(1)/downward (RingSpring clamp)
   RUNG wire#powerrail
      Contact( "DB06_Clamp".dbx0_0 )
      S_Coil( "A44" )
   END_RUNG
   // the same network as SCL:
   IF "DB06_Clamp".dbx0_0 THEN "A44" := TRUE; END_IF;
END_REGION

REGION Network 12: Welder contrast downward
   RUNG wire#powerrail
      Contact( "M2.2" )
      Contact( "Auto" )
      wire#w1
      I_Contact( "E64" )
      Coil( "DB06_Clamp".dbx0_1 )
   END_RUNG
   RUNG wire#powerrail
      Contact( "ConvOk3" )
      Contact( "DB06_Clamp".dbx4_5 )
      Contact( "Timer".T92.Q )
   END_RUNG wire#w1
   RUNG wire#powerrail
      Contact( "DB22_DisplayData".dbx16_5 )
   END_RUNG wire#w1
   RUNG wire#powerrail
      Contact( "Reset" )
      Contact( "E2.4" )
   END_RUNG wire#w1
   RUNG wire#powerrail
      Contact( "TechnoplatOk1" )
   END_RUNG wire#w1
   // the same network as SCL:
   "DB06_Clamp".dbx0_1 := (("M2.2" AND "Auto") OR ("ConvOk3" AND "DB06_Clamp".dbx4_5 AND "Timer".T92.Q) OR "DB22_DisplayData".dbx16_5 OR ("Reset" AND "E2.4") OR "TechnoplatOk1") AND NOT "E64";
END_REGION

REGION Network 13: Film clamp opening(1)/closing (RingSpring clamp)
   RUNG wire#powerrail
      Contact( "DB06_Clamp".dbx0_1 )
      I_Contact( "A50" )
      R_Coil( "A44" )
   END_RUNG
   // the same network as SCL:
   IF "DB06_Clamp".dbx0_1 AND NOT "A50" THEN "A44" := FALSE; END_IF;
END_REGION

REGION Network 14: Welder contrast forward
   "DB06_Clamp".dbx2_0 := ((("M1.0" OR "ClampCutOk8") AND "Auto") OR "DB22_DisplayData".dbx16_6) AND "Timer".T47.Q;
   "Timer".T216.TOF(IN := "DB06_Clamp".dbx2_0, PT := T#5S);   // TOF coil
END_REGION

REGION Network 15: Welder contrast forward(1)/backward (Contrast carriage)
   RUNG wire#powerrail
      Contact( "DB06_Clamp".dbx2_0 )
      wire#w1
      Coil( "A57" )
   END_RUNG
   RUNG wire#powerrail
      Contact( "Manu" )
      Contact( "Timer".T216.Q )
   END_RUNG wire#w1
   RUNG wire#w1
      R_Coil( "A58" )
   END_RUNG
   // the same network as SCL:
   "A57" := "DB06_Clamp".dbx2_0 OR ("Manu" AND "Timer".T216.Q);
   IF "A57" THEN "A58" := FALSE; END_IF;
END_REGION

REGION Network 16: Welder contrast backward
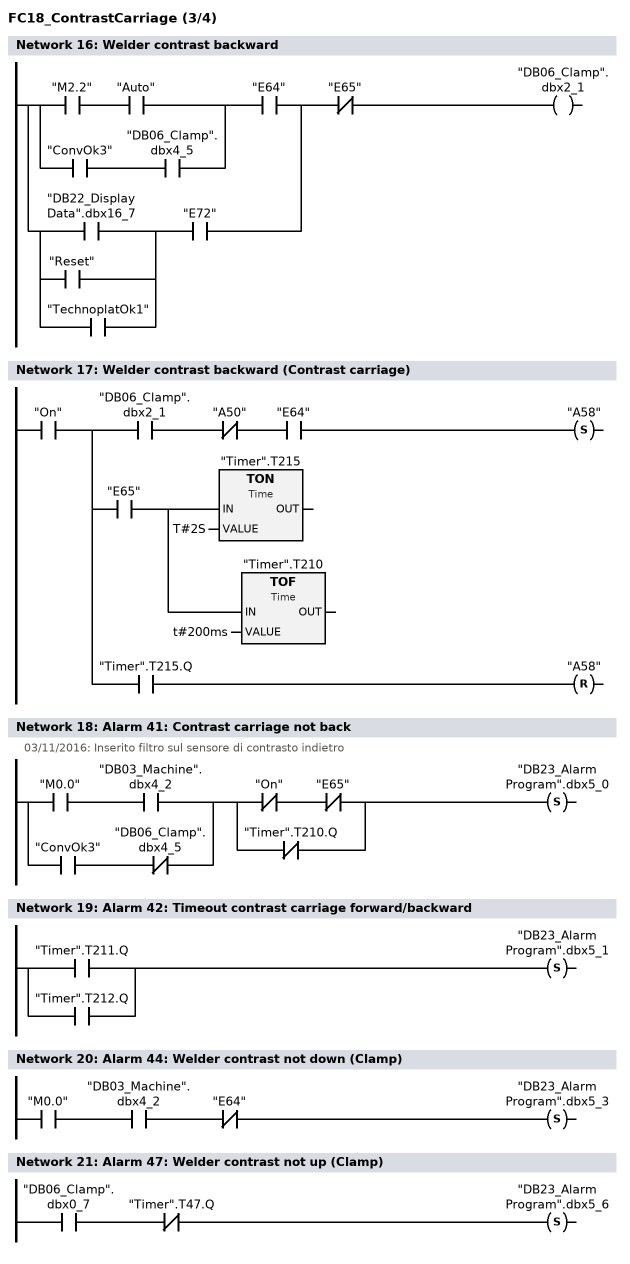
   RUNG wire#powerrail
      Contact( "M2.2" )
      Contact( "Auto" )
      wire#w1
      Contact( "E64" )
      wire#w2
      I_Contact( "E65" )
      Coil( "DB06_Clamp".dbx2_1 )
   END_RUNG
   RUNG wire#powerrail
      Contact( "ConvOk3" )
      Contact( "DB06_Clamp".dbx4_5 )
   END_RUNG wire#w1
   RUNG wire#powerrail
      Contact( "DB22_DisplayData".dbx16_7 )
      wire#w3
      Contact( "E72" )
   END_RUNG wire#w2
   RUNG wire#powerrail
      Contact( "Reset" )
   END_RUNG wire#w3
   RUNG wire#powerrail
      Contact( "TechnoplatOk1" )
   END_RUNG wire#w3
   // the same network as SCL:
   "DB06_Clamp".dbx2_1 := (((("M2.2" AND "Auto") OR ("ConvOk3" AND "DB06_Clamp".dbx4_5)) AND "E64") OR (("DB22_DisplayData".dbx16_7 OR "Reset" OR "TechnoplatOk1") AND "E72")) AND NOT "E65";
END_REGION

REGION Network 17: Welder contrast backward (Contrast carriage)
   IF "On" AND "DB06_Clamp".dbx2_1 AND NOT "A50" AND "E64" THEN "A58" := TRUE; END_IF;
   #_w1 := "On" AND "E65";
   "Timer".T215.TON(IN := #_w1, PT := T#2S);   // TON coil
   "Timer".T210.TOF(IN := #_w1, PT := t#200ms);   // TOF coil
   IF "On" AND "Timer".T215.Q THEN "A58" := FALSE; END_IF;
END_REGION

REGION Network 18: Alarm 41: Contrast carriage not back
   // 03/11/2016: Inserito filtro sul sensore di contrasto indietro
   RUNG wire#powerrail
      Contact( "M0.0" )
      Contact( "DB03_Machine".dbx4_2 )
      wire#w1
      I_Contact( "On" )
      I_Contact( "E65" )
      wire#w2
      S_Coil( "DB23_AlarmProgram".dbx5_0 )
   END_RUNG
   RUNG wire#powerrail
      Contact( "ConvOk3" )
      I_Contact( "DB06_Clamp".dbx4_5 )
   END_RUNG wire#w1
   RUNG wire#w1
      I_Contact( "Timer".T210.Q )
   END_RUNG wire#w2
   // the same network as SCL:
   IF (("M0.0" AND "DB03_Machine".dbx4_2) OR ("ConvOk3" AND NOT "DB06_Clamp".dbx4_5)) AND ((NOT "On" AND NOT "E65") OR NOT "Timer".T210.Q) THEN
       "DB23_AlarmProgram".dbx5_0 := TRUE;
   END_IF;
END_REGION

REGION Network 19: Alarm 42: Timeout contrast carriage forward/backward
   RUNG wire#powerrail
      Contact( "Timer".T211.Q )
      wire#w1
      S_Coil( "DB23_AlarmProgram".dbx5_1 )
   END_RUNG
   RUNG wire#powerrail
      Contact( "Timer".T212.Q )
   END_RUNG wire#w1
   // the same network as SCL:
   IF "Timer".T211.Q OR "Timer".T212.Q THEN "DB23_AlarmProgram".dbx5_1 := TRUE; END_IF;
END_REGION

REGION Network 20: Alarm 44: Welder contrast not down (Clamp)
   RUNG wire#powerrail
      Contact( "M0.0" )
      Contact( "DB03_Machine".dbx4_2 )
      I_Contact( "E64" )
      S_Coil( "DB23_AlarmProgram".dbx5_3 )
   END_RUNG
   // the same network as SCL:
   IF "M0.0" AND "DB03_Machine".dbx4_2 AND NOT "E64" THEN "DB23_AlarmProgram".dbx5_3 := TRUE; END_IF;
END_REGION

REGION Network 21: Alarm 47: Welder contrast not up (Clamp)
   RUNG wire#powerrail
      Contact( "DB06_Clamp".dbx0_7 )
      I_Contact( "Timer".T47.Q )
      S_Coil( "DB23_AlarmProgram".dbx5_6 )
   END_RUNG
   // the same network as SCL:
   IF "DB06_Clamp".dbx0_7 AND NOT "Timer".T47.Q THEN "DB23_AlarmProgram".dbx5_6 := TRUE; END_IF;
END_REGION

REGION Network 22: Alarm 50: Timeout for welder contrast upward/downward (Clamp)
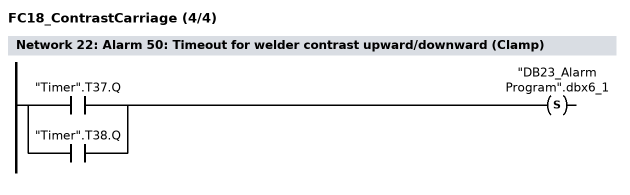
   RUNG wire#powerrail
      Contact( "Timer".T37.Q )
      wire#w1
      S_Coil( "DB23_AlarmProgram".dbx6_1 )
   END_RUNG
   RUNG wire#powerrail
      Contact( "Timer".T38.Q )
   END_RUNG wire#w1
   // the same network as SCL:
   IF "Timer".T37.Q OR "Timer".T38.Q THEN "DB23_AlarmProgram".dbx6_1 := TRUE; END_IF;
END_REGION
END_FUNCTION

FUNCTION "FC22_NoTop" : Void   // FC22, LAD
TITLE = No top
{ S7_Optimized_Access := 'FALSE' }
AUTHOR : Robopac
VERSION : 0.0
// stored: AutoNumber false, IsIECCheckEnabled false, SetENOAutomatically false, UDAEnableTagReadback false
BEGIN

REGION Network 1: TopOk10: Table rotation middle speed
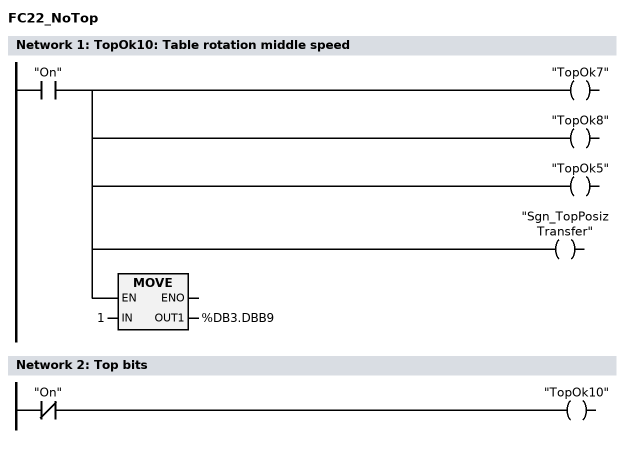
   RUNG wire#powerrail
      Contact( "On" )
      wire#w1
      Coil( "TopOk7" )
   END_RUNG
   RUNG wire#w1
      Coil( "TopOk8" )
   END_RUNG
   RUNG wire#w1
      Coil( "TopOk5" )
   END_RUNG
   RUNG wire#w1
      Coil( "Sgn_TopPosizTransfer" )
   END_RUNG
   RUNG wire#w1
      { S7_GenerateENO := "TRUE" } Move(in := 1, out1 => %DB3.DBB9)
   END_RUNG
   // the same network as SCL:
   "TopOk7" := "On";
   "TopOk8" := "On";
   "TopOk5" := "On";
   "Sgn_TopPosizTransfer" := "On";
   IF "On" THEN %DB3.DBB9 := 1; END_IF;
END_REGION

REGION Network 2: Top bits
   RUNG wire#powerrail
      I_Contact( "On" )
      Coil( "TopOk10" )
   END_RUNG
   // the same network as SCL:
   "TopOk10" := NOT "On";
END_REGION
END_FUNCTION

FUNCTION "FC23_TopTechnoplat" : Void   // FC23, LAD
TITLE = Top Inside
{ S7_Optimized_Access := 'FALSE' }
VERSION : 0.1
// stored: AutoNumber false, IsIECCheckEnabled false, SetENOAutomatically false, UDAEnableTagReadback false
   VAR_TEMP
      LW4 : Word;
   END_VAR
   VAR_TEMP   // added for the SCL form of the ladder/FBD networks
      _w1 : Bool;
      _w2 : Bool;
   END_VAR
BEGIN

REGION Network 1: Top Out Supp. Out - Signal " Top In Position for Pallet Transfe
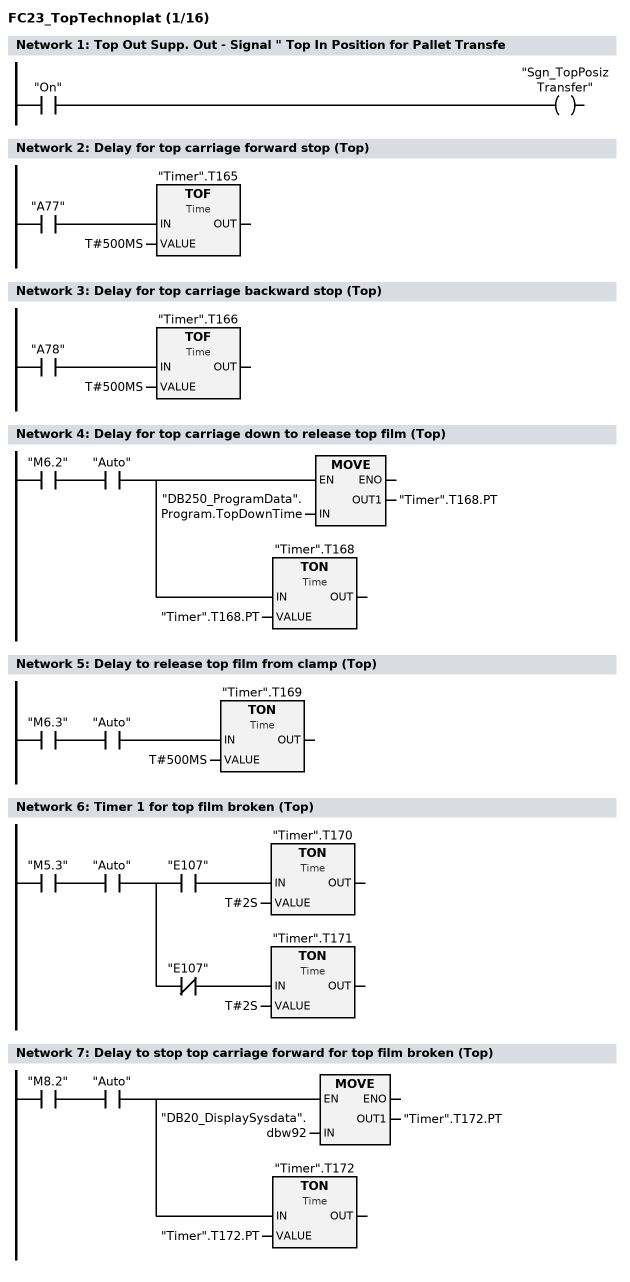
   RUNG wire#powerrail
      Contact( "On" )
      Coil( "Sgn_TopPosizTransfer" )
   END_RUNG
   // the same network as SCL:
   "Sgn_TopPosizTransfer" := "On";
END_REGION

REGION Network 2: Delay for top carriage forward stop (Top)
   "Timer".T165.TOF(IN := "A77", PT := T#500MS);   // TOF coil
END_REGION

REGION Network 3: Delay for top carriage backward stop (Top)
   "Timer".T166.TOF(IN := "A78", PT := T#500MS);   // TOF coil
END_REGION

REGION Network 4: Delay for top carriage down to release top film (Top)
   #_w1 := "M6.2" AND "Auto";
   IF #_w1 THEN "Timer".T168.PT := "DB250_ProgramData".Program.TopDownTime; END_IF;
   "Timer".T168.TON(IN := #_w1, PT := "Timer".T168.PT);   // TON coil
END_REGION

REGION Network 5: Delay to release top film from clamp (Top)
   "Timer".T169.TON(IN := "M6.3" AND "Auto", PT := T#500MS);   // TON coil
END_REGION

REGION Network 6: Timer 1 for top film broken (Top)
   #_w1 := "M5.3" AND "Auto";
   "Timer".T170.TON(IN := #_w1 AND "E107", PT := T#2S);   // TON coil
   "Timer".T171.TON(IN := #_w1 AND NOT "E107", PT := T#2S);   // TON coil
END_REGION

REGION Network 7: Delay to stop top carriage forward for top film broken (Top)
   #_w1 := "M8.2" AND "Auto";
   IF #_w1 THEN "Timer".T172.PT := "DB20_DisplaySysdata".dbw92; END_IF;
   "Timer".T172.TON(IN := #_w1, PT := "Timer".T172.PT);   // TON coil
END_REGION

REGION Network 8: Delay to stop top carriage against vibration (Top)
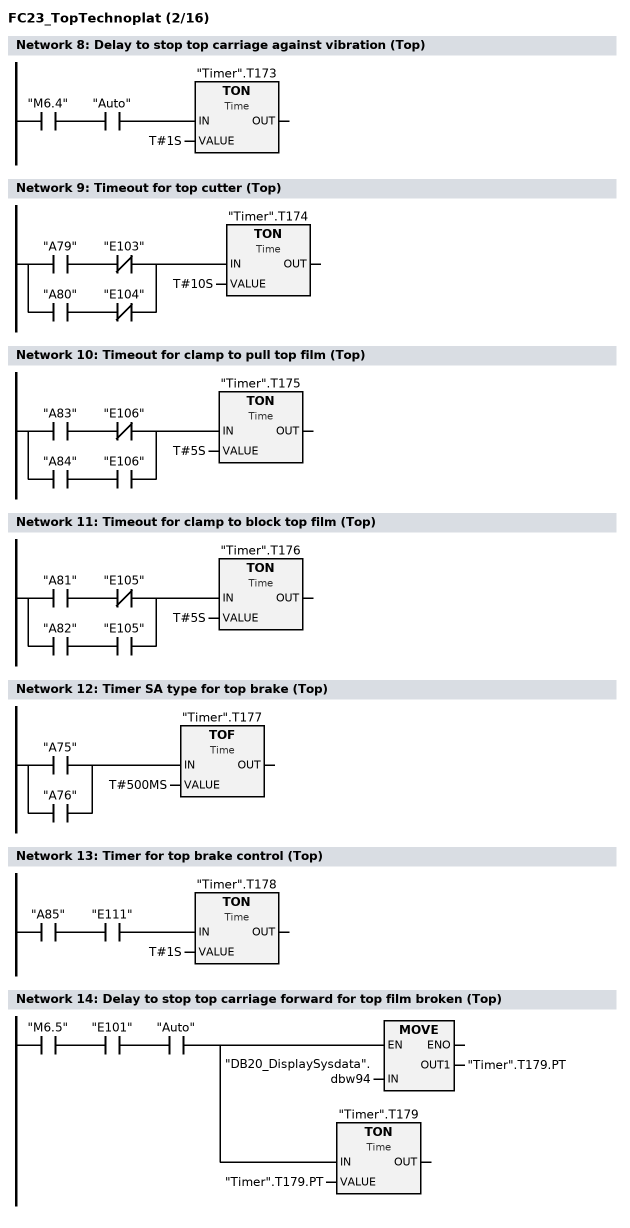
   "Timer".T173.TON(IN := "M6.4" AND "Auto", PT := T#1S);   // TON coil
END_REGION

REGION Network 9: Timeout for top cutter (Top)
   "Timer".T174.TON(IN := ("A79" AND NOT "E103") OR ("A80" AND NOT "E104"), PT := T#10S);   // TON coil
END_REGION

REGION Network 10: Timeout for clamp to pull top film (Top)
   "Timer".T175.TON(IN := ("A83" AND NOT "E106") OR ("A84" AND "E106"), PT := T#5S);   // TON coil
END_REGION

REGION Network 11: Timeout for clamp to block top film (Top)
   "Timer".T176.TON(IN := ("A81" AND NOT "E105") OR ("A82" AND "E105"), PT := T#5S);   // TON coil
END_REGION

REGION Network 12: Timer SA type for top brake (Top)
   "Timer".T177.TOF(IN := "A75" OR "A76", PT := T#500MS);   // TOF coil
END_REGION

REGION Network 13: Timer for top brake control (Top)
   "Timer".T178.TON(IN := "A85" AND "E111", PT := T#1S);   // TON coil
END_REGION

REGION Network 14: Delay to stop top carriage forward for top film broken (Top)
   #_w1 := "M6.5" AND "E101" AND "Auto";
   IF #_w1 THEN "Timer".T179.PT := "DB20_DisplaySysdata".dbw94; END_IF;
   "Timer".T179.TON(IN := #_w1, PT := "Timer".T179.PT);   // TON coil
END_REGION

REGION Network 15: Carriage in position to rotate in medium to wrap top
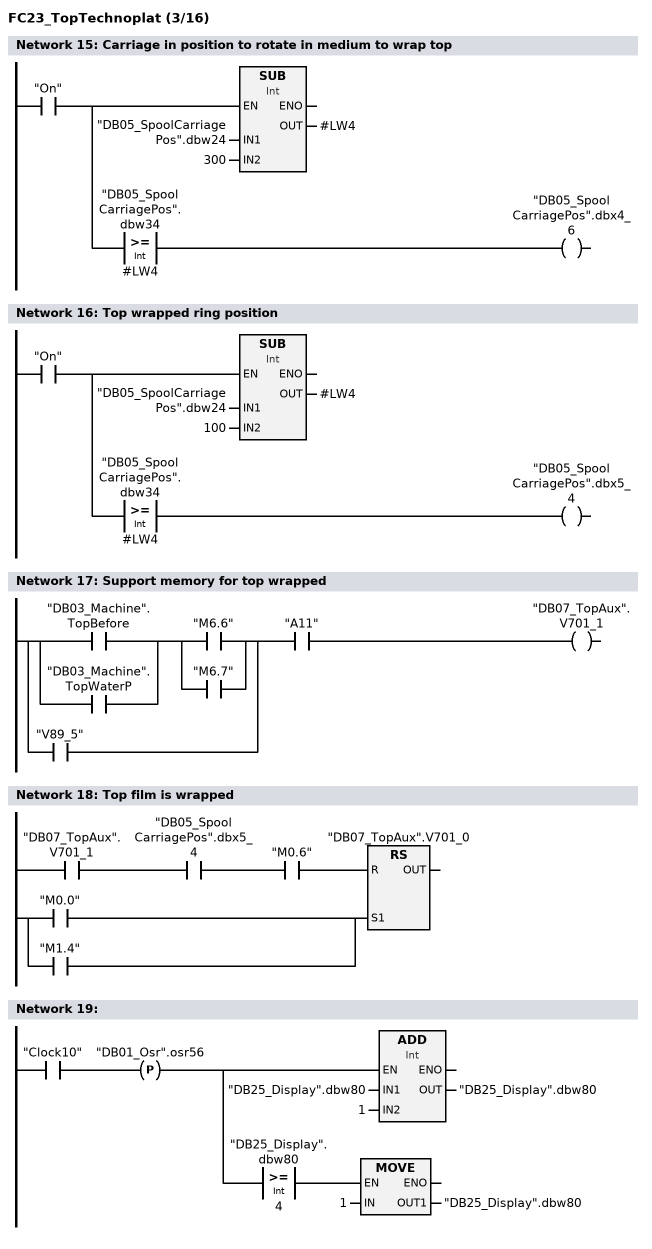
   RUNG wire#powerrail
      Contact( "On" )
      wire#w1
      { S7_Templates := "SrcType := Int"; S7_GenerateENO := "TRUE" } Sub(in1 := "DB05_SpoolCarriagePos".dbw24, in2 := 300, out => #LW4)
   END_RUNG
   RUNG wire#w1
      { S7_Templates := "SrcType := Int" } GE_Contact(in1 := "DB05_SpoolCarriagePos".dbw34, in2 := #LW4)
      Coil( "DB05_SpoolCarriagePos".dbx4_6 )
   END_RUNG
   // the same network as SCL:
   IF "On" THEN #LW4 := "DB05_SpoolCarriagePos".dbw24 - 300; END_IF;
   "DB05_SpoolCarriagePos".dbx4_6 := "On" AND ("DB05_SpoolCarriagePos".dbw34 >= #LW4);
END_REGION

REGION Network 16: Top wrapped ring position
   RUNG wire#powerrail
      Contact( "On" )
      wire#w1
      { S7_Templates := "SrcType := Int"; S7_GenerateENO := "TRUE" } Sub(in1 := "DB05_SpoolCarriagePos".dbw24, in2 := 100, out => #LW4)
   END_RUNG
   RUNG wire#w1
      { S7_Templates := "SrcType := Int" } GE_Contact(in1 := "DB05_SpoolCarriagePos".dbw34, in2 := #LW4)
      Coil( "DB05_SpoolCarriagePos".dbx5_4 )
   END_RUNG
   // the same network as SCL:
   IF "On" THEN #LW4 := "DB05_SpoolCarriagePos".dbw24 - 100; END_IF;
   "DB05_SpoolCarriagePos".dbx5_4 := "On" AND ("DB05_SpoolCarriagePos".dbw34 >= #LW4);
END_REGION

REGION Network 17: Support memory for top wrapped
   RUNG wire#powerrail
      Contact( "DB03_Machine".TopBefore )
      wire#w1
      Contact( "M6.6" )
      wire#w2
      Contact( "A11" )
      Coil( "DB07_TopAux".V701_1 )
   END_RUNG
   RUNG wire#powerrail
      Contact( "DB03_Machine".TopWaterP )
   END_RUNG wire#w1
   RUNG wire#w1
      Contact( "M6.7" )
   END_RUNG wire#w2
   RUNG wire#powerrail
      Contact( "V89_5" )
   END_RUNG wire#w2
   // the same network as SCL:
   "DB07_TopAux".V701_1 := ((("DB03_Machine".TopBefore OR "DB03_Machine".TopWaterP) AND ("M6.6" OR "M6.7")) OR "V89_5") AND "A11";
END_REGION

REGION Network 18: Top film is wrapped
   RUNG wire#powerrail
      Contact( "DB07_TopAux".V701_1 )
      Contact( "DB05_SpoolCarriagePos".dbx5_4 )
      Contact( "M0.6" )
      S_RS(operand := "DB07_TopAux".V701_0, s1 := wire#w1)
   END_RUNG
   RUNG wire#powerrail
      Contact( "M0.0" )
   END_RUNG wire#w1
   RUNG wire#powerrail
      Contact( "M1.4" )
   END_RUNG wire#w1
   // the same network as SCL:
   IF "DB07_TopAux".V701_1 AND "DB05_SpoolCarriagePos".dbx5_4 AND "M0.6" THEN
       "DB07_TopAux".V701_0 := FALSE;   // RS flip-flop
   END_IF;
   IF "M0.0" OR "M1.4" THEN "DB07_TopAux".V701_0 := TRUE; END_IF;
END_REGION

REGION Network 19
   RUNG wire#powerrail
      Contact( "Clock10" )
      P_Trig( "DB01_Osr".osr56 )
      wire#w1
      { S7_Templates := "SrcType := Int"; S7_GenerateENO := "TRUE" } Add(in1 := "DB25_Display".dbw80, in2 := 1, out => "DB25_Display".dbw80)
   END_RUNG
   RUNG wire#w1
      { S7_Templates := "SrcType := Int" } GE_Contact(in1 := "DB25_Display".dbw80, in2 := 4)
      { S7_GenerateENO := "TRUE" } Move(in := 1, out1 => "DB25_Display".dbw80)
   END_RUNG
   // the same network as SCL:
   #_w1 := "Clock10" AND NOT "DB01_Osr".osr56;   // rising edge
   "DB01_Osr".osr56 := "Clock10";
   IF #_w1 THEN "DB25_Display".dbw80 := "DB25_Display".dbw80 + 1; END_IF;
   IF #_w1 AND ("DB25_Display".dbw80 >= 4) THEN "DB25_Display".dbw80 := 1; END_IF;
END_REGION

REGION Network 20: Arm rotation speed: Middle 1 for top
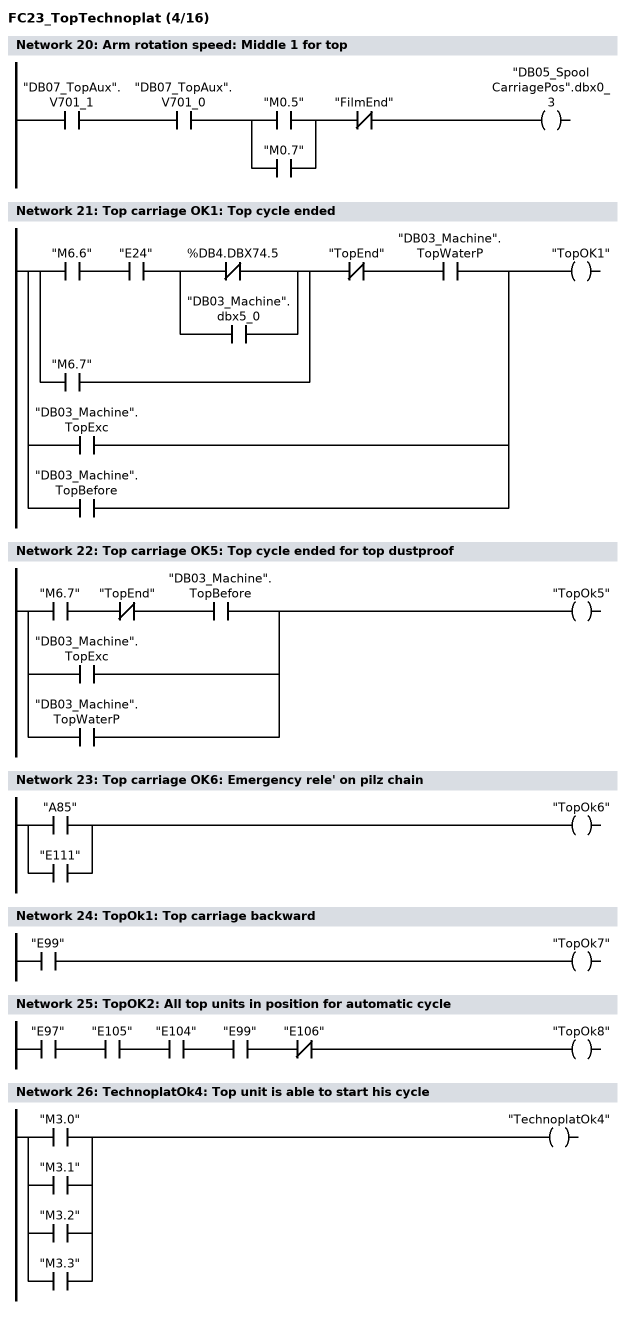
   RUNG wire#powerrail
      Contact( "DB07_TopAux".V701_1 )
      Contact( "DB07_TopAux".V701_0 )
      wire#w1
      Contact( "M0.5" )
      wire#w2
      I_Contact( "FilmEnd" )
      Coil( "DB05_SpoolCarriagePos".dbx0_3 )
   END_RUNG
   RUNG wire#w1
      Contact( "M0.7" )
   END_RUNG wire#w2
   // the same network as SCL:
   "DB05_SpoolCarriagePos".dbx0_3 := "DB07_TopAux".V701_1 AND "DB07_TopAux".V701_0 AND ("M0.5" OR "M0.7") AND NOT "FilmEnd";
END_REGION

REGION Network 21: Top carriage OK1: Top cycle ended
   RUNG wire#powerrail
      Contact( "M6.6" )
      Contact( "E24" )
      wire#w1
      I_Contact( %DB4.DBX74.5 )
      wire#w2
      I_Contact( "TopEnd" )
      Contact( "DB03_Machine".TopWaterP )
      wire#w3
      Coil( "TopOK1" )
   END_RUNG
   RUNG wire#w1
      Contact( "DB03_Machine".dbx5_0 )
   END_RUNG wire#w2
   RUNG wire#powerrail
      Contact( "M6.7" )
   END_RUNG wire#w2
   RUNG wire#powerrail
      Contact( "DB03_Machine".TopExc )
   END_RUNG wire#w3
   RUNG wire#powerrail
      Contact( "DB03_Machine".TopBefore )
   END_RUNG wire#w3
   // the same network as SCL:
   "TopOK1" := ((("M6.6" AND "E24" AND (NOT %DB4.DBX74.5 OR "DB03_Machine".dbx5_0)) OR "M6.7") AND NOT "TopEnd" AND "DB03_Machine".TopWaterP) OR "DB03_Machine".TopExc OR "DB03_Machine".TopBefore;
END_REGION

REGION Network 22: Top carriage OK5: Top cycle ended for top dustproof
   RUNG wire#powerrail
      Contact( "M6.7" )
      I_Contact( "TopEnd" )
      Contact( "DB03_Machine".TopBefore )
      wire#w1
      Coil( "TopOk5" )
   END_RUNG
   RUNG wire#powerrail
      Contact( "DB03_Machine".TopExc )
   END_RUNG wire#w1
   RUNG wire#powerrail
      Contact( "DB03_Machine".TopWaterP )
   END_RUNG wire#w1
   // the same network as SCL:
   "TopOk5" := ("M6.7" AND NOT "TopEnd" AND "DB03_Machine".TopBefore) OR "DB03_Machine".TopExc OR "DB03_Machine".TopWaterP;
END_REGION

REGION Network 23: Top carriage OK6: Emergency rele' on pilz chain
   RUNG wire#powerrail
      Contact( "A85" )
      wire#w1
      Coil( "TopOk6" )
   END_RUNG
   RUNG wire#powerrail
      Contact( "E111" )
   END_RUNG wire#w1
   // the same network as SCL:
   "TopOk6" := "A85" OR "E111";
END_REGION

REGION Network 24: TopOk1: Top carriage backward
   RUNG wire#powerrail
      Contact( "E99" )
      Coil( "TopOk7" )
   END_RUNG
   // the same network as SCL:
   "TopOk7" := "E99";
END_REGION

REGION Network 25: TopOK2: All top units in position for automatic cycle
   RUNG wire#powerrail
      Contact( "E97" )
      Contact( "E105" )
      Contact( "E104" )
      Contact( "E99" )
      I_Contact( "E106" )
      Coil( "TopOk8" )
   END_RUNG
   // the same network as SCL:
   "TopOk8" := "E97" AND "E105" AND "E104" AND "E99" AND NOT "E106";
END_REGION

REGION Network 26: TechnoplatOk4: Top unit is able to start his cycle
   RUNG wire#powerrail
      Contact( "M3.0" )
      wire#w1
      Coil( "TechnoplatOk4" )
   END_RUNG
   RUNG wire#powerrail
      Contact( "M3.1" )
   END_RUNG wire#w1
   RUNG wire#powerrail
      Contact( "M3.2" )
   END_RUNG wire#w1
   RUNG wire#powerrail
      Contact( "M3.3" )
   END_RUNG wire#w1
   // the same network as SCL:
   "TechnoplatOk4" := "M3.0" OR "M3.1" OR "M3.2" OR "M3.3";
END_REGION

REGION Network 27: Top film ended or broken
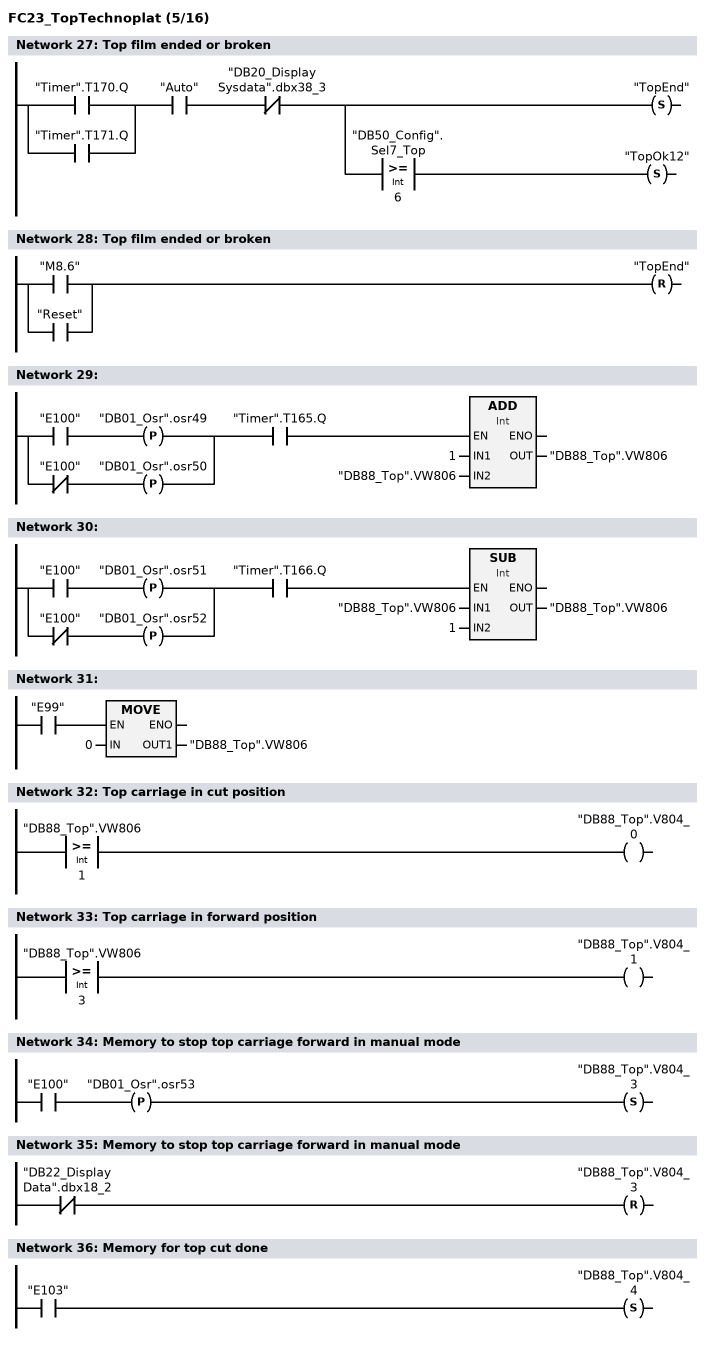
   RUNG wire#powerrail
      Contact( "Timer".T170.Q )
      wire#w1
      Contact( "Auto" )
      I_Contact( "DB20_DisplaySysdata".dbx38_3 )
      wire#w2
      S_Coil( "TopEnd" )
   END_RUNG
   RUNG wire#powerrail
      Contact( "Timer".T171.Q )
   END_RUNG wire#w1
   RUNG wire#w2
      { S7_Templates := "SrcType := Int" } GE_Contact(in1 := "DB50_Config".Sel7_Top, in2 := 6)
      S_Coil( "TopOk12" )
   END_RUNG
   // the same network as SCL:
   #_w1 := ("Timer".T170.Q OR "Timer".T171.Q) AND "Auto" AND NOT "DB20_DisplaySysdata".dbx38_3;
   IF #_w1 THEN "TopEnd" := TRUE; END_IF;
   IF #_w1 AND ("DB50_Config".Sel7_Top >= 6) THEN "TopOk12" := TRUE; END_IF;
END_REGION

REGION Network 28: Top film ended or broken
   RUNG wire#powerrail
      Contact( "M8.6" )
      wire#w1
      R_Coil( "TopEnd" )
   END_RUNG
   RUNG wire#powerrail
      Contact( "Reset" )
   END_RUNG wire#w1
   // the same network as SCL:
   IF "M8.6" OR "Reset" THEN "TopEnd" := FALSE; END_IF;
END_REGION

REGION Network 29
   RUNG wire#powerrail
      Contact( "E100" )
      P_Trig( "DB01_Osr".osr49 )
      wire#w1
      Contact( "Timer".T165.Q )
      { S7_Templates := "SrcType := Int"; S7_GenerateENO := "TRUE" } Add(in1 := 1, in2 := "DB88_Top".VW806, out => "DB88_Top".VW806)
   END_RUNG
   RUNG wire#powerrail
      I_Contact( "E100" )
      P_Trig( "DB01_Osr".osr50 )
   END_RUNG wire#w1
   // the same network as SCL:
   #_w1 := "E100" AND NOT "DB01_Osr".osr49;   // rising edge
   "DB01_Osr".osr49 := "E100";
   #_w2 := NOT "E100" AND NOT "DB01_Osr".osr50;   // rising edge
   "DB01_Osr".osr50 := NOT "E100";
   IF (#_w1 OR #_w2) AND "Timer".T165.Q THEN "DB88_Top".VW806 := 1 + "DB88_Top".VW806; END_IF;
END_REGION

REGION Network 30
   RUNG wire#powerrail
      Contact( "E100" )
      P_Trig( "DB01_Osr".osr51 )
      wire#w1
      Contact( "Timer".T166.Q )
      { S7_Templates := "SrcType := Int"; S7_GenerateENO := "TRUE" } Sub(in1 := "DB88_Top".VW806, in2 := 1, out => "DB88_Top".VW806)
   END_RUNG
   RUNG wire#powerrail
      I_Contact( "E100" )
      P_Trig( "DB01_Osr".osr52 )
   END_RUNG wire#w1
   // the same network as SCL:
   #_w1 := "E100" AND NOT "DB01_Osr".osr51;   // rising edge
   "DB01_Osr".osr51 := "E100";
   #_w2 := NOT "E100" AND NOT "DB01_Osr".osr52;   // rising edge
   "DB01_Osr".osr52 := NOT "E100";
   IF (#_w1 OR #_w2) AND "Timer".T166.Q THEN "DB88_Top".VW806 := "DB88_Top".VW806 - 1; END_IF;
END_REGION

REGION Network 31
   RUNG wire#powerrail
      Contact( "E99" )
      { S7_GenerateENO := "TRUE" } Move(in := 0, out1 => "DB88_Top".VW806)
   END_RUNG
   // the same network as SCL:
   IF "E99" THEN "DB88_Top".VW806 := 0; END_IF;
END_REGION

REGION Network 32: Top carriage in cut position
   RUNG wire#powerrail
      { S7_Templates := "SrcType := Int" } GE_Contact(in1 := "DB88_Top".VW806, in2 := 1)
      Coil( "DB88_Top".V804_0 )
   END_RUNG
   // the same network as SCL:
   "DB88_Top".V804_0 := "DB88_Top".VW806 >= 1;
END_REGION

REGION Network 33: Top carriage in forward position
   RUNG wire#powerrail
      { S7_Templates := "SrcType := Int" } GE_Contact(in1 := "DB88_Top".VW806, in2 := 3)
      Coil( "DB88_Top".V804_1 )
   END_RUNG
   // the same network as SCL:
   "DB88_Top".V804_1 := "DB88_Top".VW806 >= 3;
END_REGION

REGION Network 34: Memory to stop top carriage forward in manual mode
   RUNG wire#powerrail
      Contact( "E100" )
      P_Trig( "DB01_Osr".osr53 )
      S_Coil( "DB88_Top".V804_3 )
   END_RUNG
   // the same network as SCL:
   #_w1 := "E100" AND NOT "DB01_Osr".osr53;   // rising edge
   "DB01_Osr".osr53 := "E100";
   IF #_w1 THEN "DB88_Top".V804_3 := TRUE; END_IF;
END_REGION

REGION Network 35: Memory to stop top carriage forward in manual mode
   RUNG wire#powerrail
      I_Contact( "DB22_DisplayData".dbx18_2 )
      R_Coil( "DB88_Top".V804_3 )
   END_RUNG
   // the same network as SCL:
   IF NOT "DB22_DisplayData".dbx18_2 THEN "DB88_Top".V804_3 := FALSE; END_IF;
END_REGION

REGION Network 36: Memory for top cut done
   RUNG wire#powerrail
      Contact( "E103" )
      S_Coil( "DB88_Top".V804_4 )
   END_RUNG
   // the same network as SCL:
   IF "E103" THEN "DB88_Top".V804_4 := TRUE; END_IF;
END_REGION

REGION Network 37: Memory for top cut done
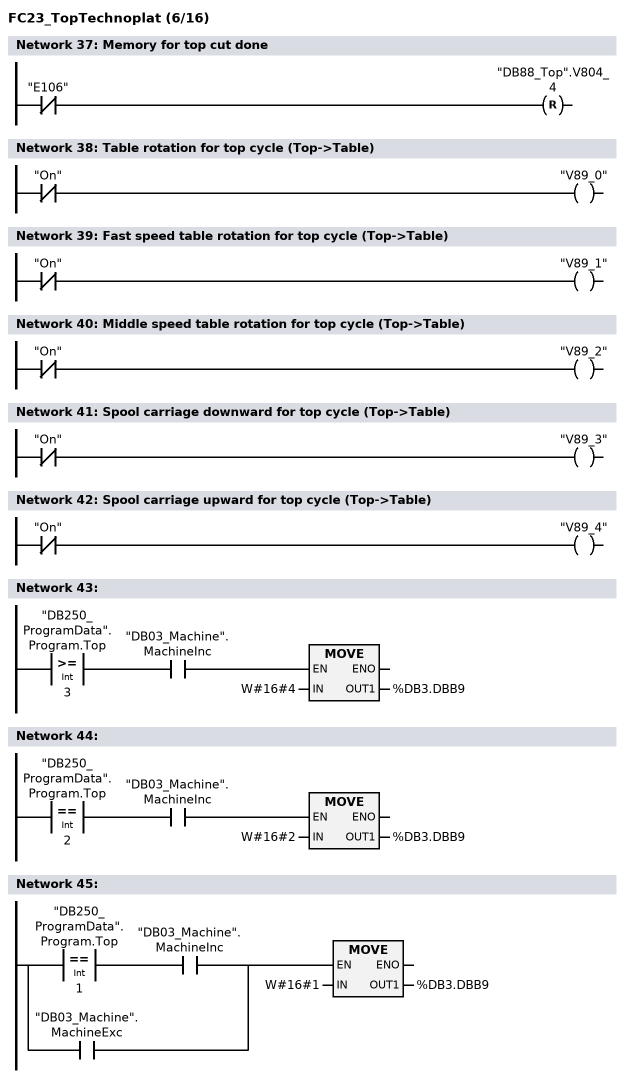
   RUNG wire#powerrail
      I_Contact( "E106" )
      R_Coil( "DB88_Top".V804_4 )
   END_RUNG
   // the same network as SCL:
   IF NOT "E106" THEN "DB88_Top".V804_4 := FALSE; END_IF;
END_REGION

REGION Network 38: Table rotation for top cycle (Top->Table)
   RUNG wire#powerrail
      I_Contact( "On" )
      Coil( "V89_0" )
   END_RUNG
   // the same network as SCL:
   "V89_0" := NOT "On";
END_REGION

REGION Network 39: Fast speed table rotation for top cycle (Top->Table)
   RUNG wire#powerrail
      I_Contact( "On" )
      Coil( "V89_1" )
   END_RUNG
   // the same network as SCL:
   "V89_1" := NOT "On";
END_REGION

REGION Network 40: Middle speed table rotation for top cycle (Top->Table)
   RUNG wire#powerrail
      I_Contact( "On" )
      Coil( "V89_2" )
   END_RUNG
   // the same network as SCL:
   "V89_2" := NOT "On";
END_REGION

REGION Network 41: Spool carriage downward for top cycle (Top->Table)
   RUNG wire#powerrail
      I_Contact( "On" )
      Coil( "V89_3" )
   END_RUNG
   // the same network as SCL:
   "V89_3" := NOT "On";
END_REGION

REGION Network 42: Spool carriage upward for top cycle (Top->Table)
   RUNG wire#powerrail
      I_Contact( "On" )
      Coil( "V89_4" )
   END_RUNG
   // the same network as SCL:
   "V89_4" := NOT "On";
END_REGION

REGION Network 43
   RUNG wire#powerrail
      { S7_Templates := "SrcType := Int" } GE_Contact(in1 := "DB250_ProgramData".Program.Top, in2 := 3)
      Contact( "DB03_Machine".MachineInc )
      { S7_GenerateENO := "TRUE" } Move(in := W#16#4, out1 => %DB3.DBB9)
   END_RUNG
   // the same network as SCL:
   IF ("DB250_ProgramData".Program.Top >= 3) AND "DB03_Machine".MachineInc THEN %DB3.DBB9 := W#16#4; END_IF;
END_REGION

REGION Network 44
   RUNG wire#powerrail
      { S7_Templates := "SrcType := Int" } EQ_Contact(in1 := "DB250_ProgramData".Program.Top, in2 := 2)
      Contact( "DB03_Machine".MachineInc )
      { S7_GenerateENO := "TRUE" } Move(in := W#16#2, out1 => %DB3.DBB9)
   END_RUNG
   // the same network as SCL:
   IF ("DB250_ProgramData".Program.Top = 2) AND "DB03_Machine".MachineInc THEN %DB3.DBB9 := W#16#2; END_IF;
END_REGION

REGION Network 45
   RUNG wire#powerrail
      { S7_Templates := "SrcType := Int" } EQ_Contact(in1 := "DB250_ProgramData".Program.Top, in2 := 1)
      Contact( "DB03_Machine".MachineInc )
      wire#w1
      { S7_GenerateENO := "TRUE" } Move(in := W#16#1, out1 => %DB3.DBB9)
   END_RUNG
   RUNG wire#powerrail
      Contact( "DB03_Machine".MachineExc )
   END_RUNG wire#w1
   // the same network as SCL:
   IF (("DB250_ProgramData".Program.Top = 1) AND "DB03_Machine".MachineInc) OR "DB03_Machine".MachineExc THEN
       %DB3.DBB9 := W#16#1;
   END_IF;
END_REGION

REGION Network 46: Wrapping cycle: After this step top waterproof
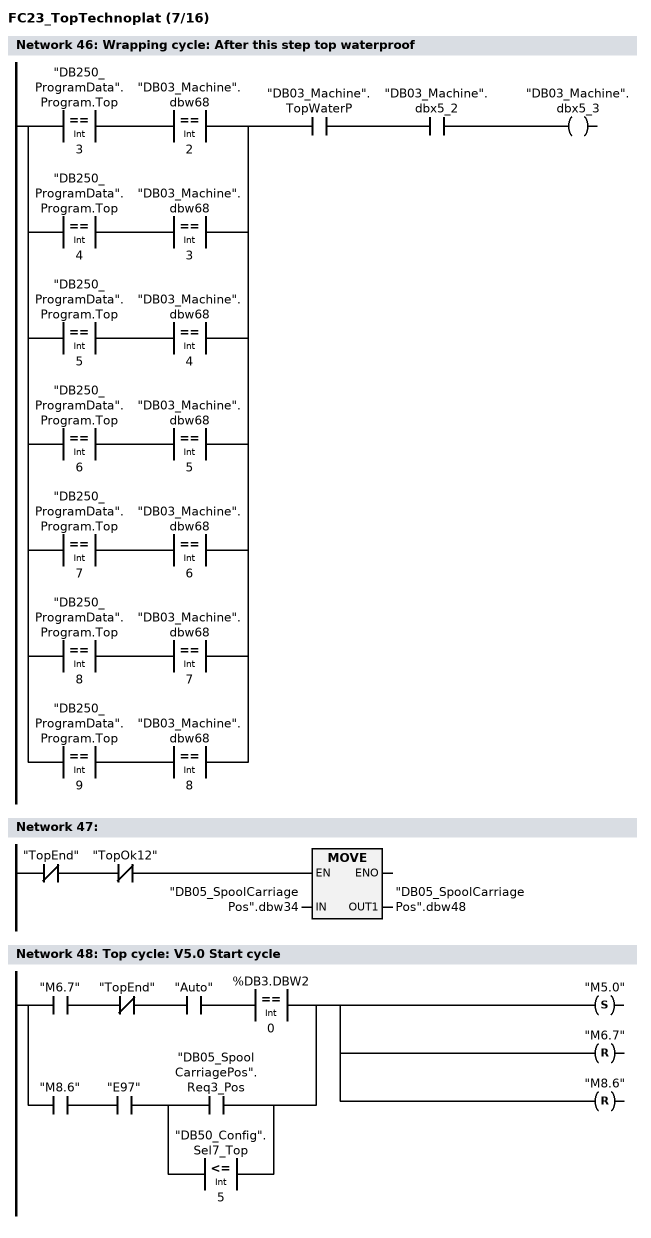
   RUNG wire#powerrail
      { S7_Templates := "SrcType := Int" } EQ_Contact(in1 := "DB250_ProgramData".Program.Top, in2 := 3)
      { S7_Templates := "SrcType := Int" } EQ_Contact(in1 := "DB03_Machine".dbw68, in2 := 2)
      wire#w1
      Contact( "DB03_Machine".TopWaterP )
      Contact( "DB03_Machine".dbx5_2 )
      Coil( "DB03_Machine".dbx5_3 )
   END_RUNG
   RUNG wire#powerrail
      { S7_Templates := "SrcType := Int" } EQ_Contact(in1 := "DB250_ProgramData".Program.Top, in2 := 4)
      { S7_Templates := "SrcType := Int" } EQ_Contact(in1 := "DB03_Machine".dbw68, in2 := 3)
   END_RUNG wire#w1
   RUNG wire#powerrail
      { S7_Templates := "SrcType := Int" } EQ_Contact(in1 := "DB250_ProgramData".Program.Top, in2 := 5)
      { S7_Templates := "SrcType := Int" } EQ_Contact(in1 := "DB03_Machine".dbw68, in2 := 4)
   END_RUNG wire#w1
   RUNG wire#powerrail
      { S7_Templates := "SrcType := Int" } EQ_Contact(in1 := "DB250_ProgramData".Program.Top, in2 := 6)
      { S7_Templates := "SrcType := Int" } EQ_Contact(in1 := "DB03_Machine".dbw68, in2 := 5)
   END_RUNG wire#w1
   RUNG wire#powerrail
      { S7_Templates := "SrcType := Int" } EQ_Contact(in1 := "DB250_ProgramData".Program.Top, in2 := 7)
      { S7_Templates := "SrcType := Int" } EQ_Contact(in1 := "DB03_Machine".dbw68, in2 := 6)
   END_RUNG wire#w1
   RUNG wire#powerrail
      { S7_Templates := "SrcType := Int" } EQ_Contact(in1 := "DB250_ProgramData".Program.Top, in2 := 8)
      { S7_Templates := "SrcType := Int" } EQ_Contact(in1 := "DB03_Machine".dbw68, in2 := 7)
   END_RUNG wire#w1
   RUNG wire#powerrail
      { S7_Templates := "SrcType := Int" } EQ_Contact(in1 := "DB250_ProgramData".Program.Top, in2 := 9)
      { S7_Templates := "SrcType := Int" } EQ_Contact(in1 := "DB03_Machine".dbw68, in2 := 8)
   END_RUNG wire#w1
   // the same network as SCL:
   "DB03_Machine".dbx5_3 := ((("DB250_ProgramData".Program.Top = 3) AND ("DB03_Machine".dbw68 = 2)) OR (("DB250_ProgramData".Program.Top = 4) AND ("DB03_Machine".dbw68 = 3)) OR (("DB250_ProgramData".Program.Top = 5) AND ("DB03_Machine".dbw68 = 4)) OR (("DB250_ProgramData".Program.Top = 6) AND ("DB03_Machine".dbw68 = 5)) OR (("DB250_ProgramData".Program.Top = 7) AND ("DB03_Machine".dbw68 = 6)) OR (("DB250_ProgramData".Program.Top = 8) AND ("DB03_Machine".dbw68 = 7)) OR (("DB250_ProgramData".Program.Top = 9) AND ("DB03_Machine".dbw68 = 8))) AND "DB03_Machine".TopWaterP AND "DB03_Machine".dbx5_2;
END_REGION

REGION Network 47
   RUNG wire#powerrail
      I_Contact( "TopEnd" )
      I_Contact( "TopOk12" )
      { S7_GenerateENO := "TRUE" } Move(in := "DB05_SpoolCarriagePos".dbw34, out1 => "DB05_SpoolCarriagePos".dbw48)
   END_RUNG
   // the same network as SCL:
   IF NOT "TopEnd" AND NOT "TopOk12" THEN
       "DB05_SpoolCarriagePos".dbw48 := "DB05_SpoolCarriagePos".dbw34;
   END_IF;
END_REGION

REGION Network 48: Top cycle: V5.0 Start cycle
   RUNG wire#powerrail
      Contact( "M6.7" )
      I_Contact( "TopEnd" )
      Contact( "Auto" )
      { S7_Templates := "SrcType := Int" } EQ_Contact(in1 := %DB3.DBW2, in2 := 0)
      wire#w1
      S_Coil( "M5.0" )
   END_RUNG
   RUNG wire#powerrail
      Contact( "M8.6" )
      Contact( "E97" )
      wire#w2
      Contact( "DB05_SpoolCarriagePos".Req3_Pos )
   END_RUNG wire#w1
   RUNG wire#w2
      { S7_Templates := "SrcType := Int" } LE_Contact(in1 := "DB50_Config".Sel7_Top, in2 := 5)
   END_RUNG wire#w1
   RUNG wire#w1
      R_Coil( "M6.7" )
   END_RUNG
   RUNG wire#w1
      R_Coil( "M8.6" )
   END_RUNG
   // the same network as SCL:
   IF ("M6.7" AND NOT "TopEnd" AND "Auto" AND (%DB3.DBW2 = 0)) OR ("M8.6" AND "E97" AND ("DB05_SpoolCarriagePos".Req3_Pos OR ("DB50_Config".Sel7_Top <= 5))) THEN
       "M5.0" := TRUE;
   END_IF;
   #_w1 := ("M6.7" AND NOT "TopEnd" AND "Auto" AND (%DB3.DBW2 = 0)) OR ("M8.6" AND "E97" AND ("DB05_SpoolCarriagePos".Req3_Pos OR ("DB50_Config".Sel7_Top <= 5)));
   IF #_w1 THEN
       "M6.7" := FALSE;
       "M8.6" := FALSE;
   END_IF;
END_REGION

REGION Network 49: Top cycle: V5.1 Closing clamp to pull top film
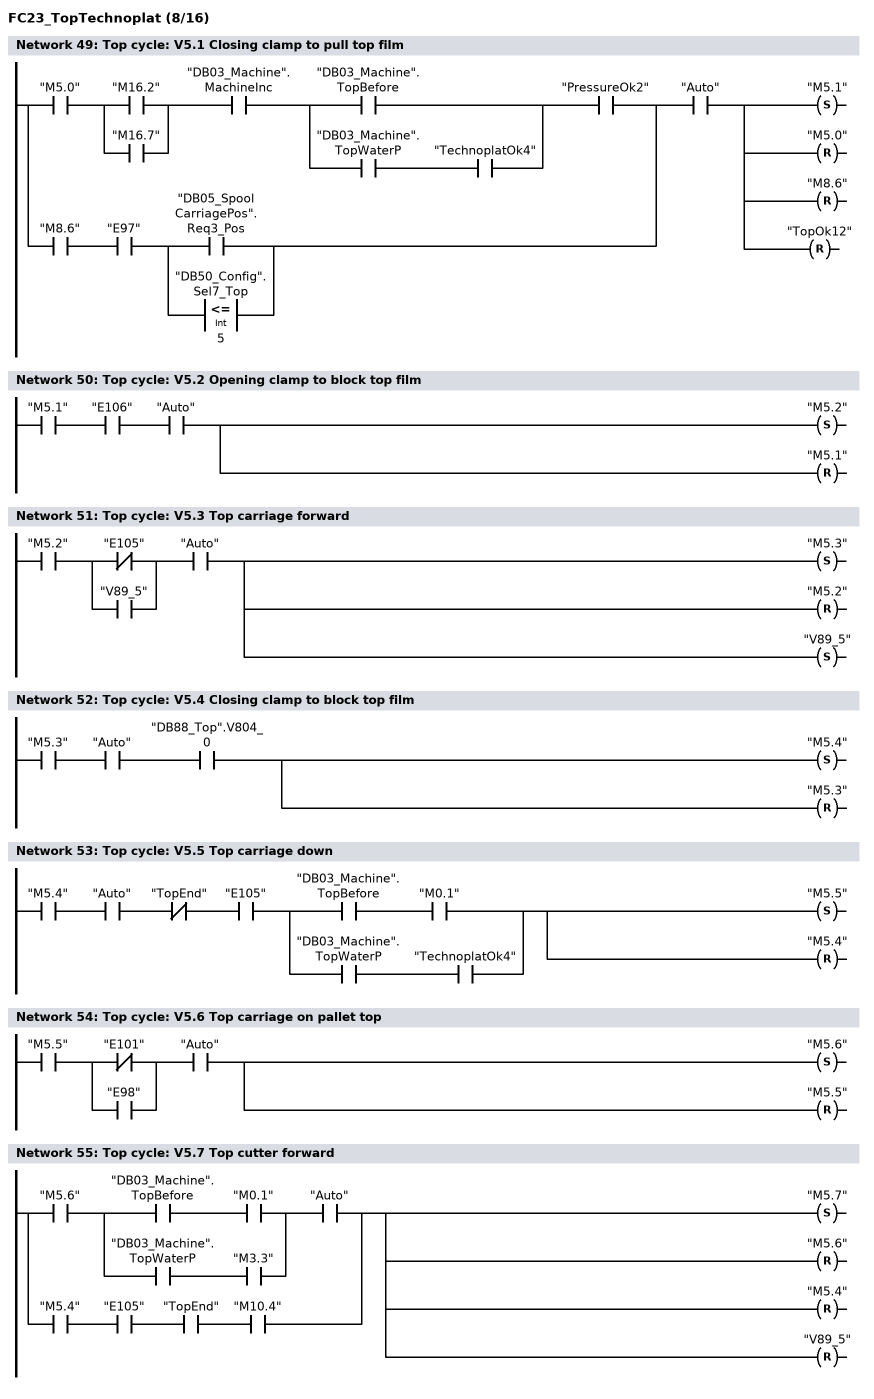
   RUNG wire#powerrail
      Contact( "M5.0" )
      wire#w1
      Contact( "M16.2" )
      wire#w2
      Contact( "DB03_Machine".MachineInc )
      wire#w3
      Contact( "DB03_Machine".TopBefore )
      wire#w4
      Contact( "PressureOk2" )
      wire#w5
      Contact( "Auto" )
      wire#w7
      S_Coil( "M5.1" )
   END_RUNG
   RUNG wire#w1
      Contact( "M16.7" )
   END_RUNG wire#w2
   RUNG wire#w3
      Contact( "DB03_Machine".TopWaterP )
      Contact( "TechnoplatOk4" )
   END_RUNG wire#w4
   RUNG wire#powerrail
      Contact( "M8.6" )
      Contact( "E97" )
      wire#w6
      Contact( "DB05_SpoolCarriagePos".Req3_Pos )
   END_RUNG wire#w5
   RUNG wire#w6
      { S7_Templates := "SrcType := Int" } LE_Contact(in1 := "DB50_Config".Sel7_Top, in2 := 5)
   END_RUNG wire#w5
   RUNG wire#w7
      R_Coil( "M5.0" )
   END_RUNG
   RUNG wire#w7
      R_Coil( "M8.6" )
   END_RUNG
   RUNG wire#w7
      R_Coil( "TopOk12" )
   END_RUNG
   // the same network as SCL:
   IF (("M5.0" AND ("M16.2" OR "M16.7") AND "DB03_Machine".MachineInc AND ("DB03_Machine".TopBefore OR ("DB03_Machine".TopWaterP AND "TechnoplatOk4")) AND "PressureOk2") OR ("M8.6" AND "E97" AND ("DB05_SpoolCarriagePos".Req3_Pos OR ("DB50_Config".Sel7_Top <= 5)))) AND "Auto" THEN
       "M5.1" := TRUE;
   END_IF;
   #_w1 := (("M5.0" AND ("M16.2" OR "M16.7") AND "DB03_Machine".MachineInc AND ("DB03_Machine".TopBefore OR ("DB03_Machine".TopWaterP AND "TechnoplatOk4")) AND "PressureOk2") OR ("M8.6" AND "E97" AND ("DB05_SpoolCarriagePos".Req3_Pos OR ("DB50_Config".Sel7_Top <= 5)))) AND "Auto";
   IF #_w1 THEN
       "M5.0" := FALSE;
       "M8.6" := FALSE;
       "TopOk12" := FALSE;
   END_IF;
END_REGION

REGION Network 50: Top cycle: V5.2 Opening clamp to block top film
   RUNG wire#powerrail
      Contact( "M5.1" )
      Contact( "E106" )
      Contact( "Auto" )
      wire#w1
      S_Coil( "M5.2" )
   END_RUNG
   RUNG wire#w1
      R_Coil( "M5.1" )
   END_RUNG
   // the same network as SCL:
   IF "M5.1" AND "E106" AND "Auto" THEN
       "M5.2" := TRUE;
       "M5.1" := FALSE;
   END_IF;
END_REGION

REGION Network 51: Top cycle: V5.3 Top carriage forward
   RUNG wire#powerrail
      Contact( "M5.2" )
      wire#w1
      I_Contact( "E105" )
      wire#w2
      Contact( "Auto" )
      wire#w3
      S_Coil( "M5.3" )
   END_RUNG
   RUNG wire#w1
      Contact( "V89_5" )
   END_RUNG wire#w2
   RUNG wire#w3
      R_Coil( "M5.2" )
   END_RUNG
   RUNG wire#w3
      S_Coil( "V89_5" )
   END_RUNG
   // the same network as SCL:
   IF "M5.2" AND (NOT "E105" OR "V89_5") AND "Auto" THEN "M5.3" := TRUE; END_IF;
   #_w1 := "M5.2" AND (NOT "E105" OR "V89_5") AND "Auto";
   IF #_w1 THEN
       "M5.2" := FALSE;
       "V89_5" := TRUE;
   END_IF;
END_REGION

REGION Network 52: Top cycle: V5.4 Closing clamp to block top film
   RUNG wire#powerrail
      Contact( "M5.3" )
      Contact( "Auto" )
      Contact( "DB88_Top".V804_0 )
      wire#w1
      S_Coil( "M5.4" )
   END_RUNG
   RUNG wire#w1
      R_Coil( "M5.3" )
   END_RUNG
   // the same network as SCL:
   IF "M5.3" AND "Auto" AND "DB88_Top".V804_0 THEN
       "M5.4" := TRUE;
       "M5.3" := FALSE;
   END_IF;
END_REGION

REGION Network 53: Top cycle: V5.5 Top carriage down
   RUNG wire#powerrail
      Contact( "M5.4" )
      Contact( "Auto" )
      I_Contact( "TopEnd" )
      Contact( "E105" )
      wire#w1
      Contact( "DB03_Machine".TopBefore )
      Contact( "M0.1" )
      wire#w2
      S_Coil( "M5.5" )
   END_RUNG
   RUNG wire#w1
      Contact( "DB03_Machine".TopWaterP )
      Contact( "TechnoplatOk4" )
   END_RUNG wire#w2
   RUNG wire#w2
      R_Coil( "M5.4" )
   END_RUNG
   // the same network as SCL:
   IF "M5.4" AND "Auto" AND NOT "TopEnd" AND "E105" AND (("DB03_Machine".TopBefore AND "M0.1") OR ("DB03_Machine".TopWaterP AND "TechnoplatOk4")) THEN
       "M5.5" := TRUE;
       "M5.4" := FALSE;
   END_IF;
END_REGION

REGION Network 54: Top cycle: V5.6 Top carriage on pallet top
   RUNG wire#powerrail
      Contact( "M5.5" )
      wire#w1
      I_Contact( "E101" )
      wire#w2
      Contact( "Auto" )
      wire#w3
      S_Coil( "M5.6" )
   END_RUNG
   RUNG wire#w1
      Contact( "E98" )
   END_RUNG wire#w2
   RUNG wire#w3
      R_Coil( "M5.5" )
   END_RUNG
   // the same network as SCL:
   IF "M5.5" AND (NOT "E101" OR "E98") AND "Auto" THEN
       "M5.6" := TRUE;
       "M5.5" := FALSE;
   END_IF;
END_REGION

REGION Network 55: Top cycle: V5.7 Top cutter forward
   RUNG wire#powerrail
      Contact( "M5.6" )
      wire#w1
      Contact( "DB03_Machine".TopBefore )
      Contact( "M0.1" )
      wire#w2
      Contact( "Auto" )
      wire#w3
      S_Coil( "M5.7" )
   END_RUNG
   RUNG wire#w1
      Contact( "DB03_Machine".TopWaterP )
      Contact( "M3.3" )
   END_RUNG wire#w2
   RUNG wire#powerrail
      Contact( "M5.4" )
      Contact( "E105" )
      Contact( "TopEnd" )
      Contact( "M10.4" )
   END_RUNG wire#w3
   RUNG wire#w3
      R_Coil( "M5.6" )
   END_RUNG
   RUNG wire#w3
      R_Coil( "M5.4" )
   END_RUNG
   RUNG wire#w3
      R_Coil( "V89_5" )
   END_RUNG
   // the same network as SCL:
   IF ("M5.6" AND (("DB03_Machine".TopBefore AND "M0.1") OR ("DB03_Machine".TopWaterP AND "M3.3")) AND "Auto") OR ("M5.4" AND "E105" AND "TopEnd" AND "M10.4") THEN
       "M5.7" := TRUE;
   END_IF;
   #_w1 := ("M5.6" AND (("DB03_Machine".TopBefore AND "M0.1") OR ("DB03_Machine".TopWaterP AND "M3.3")) AND "Auto") OR ("M5.4" AND "E105" AND "TopEnd" AND "M10.4");
   IF #_w1 THEN
       "M5.6" := FALSE;
       "M5.4" := FALSE;
       "V89_5" := FALSE;
   END_IF;
END_REGION

REGION Network 56: Top cycle: M6.0 Start cycle
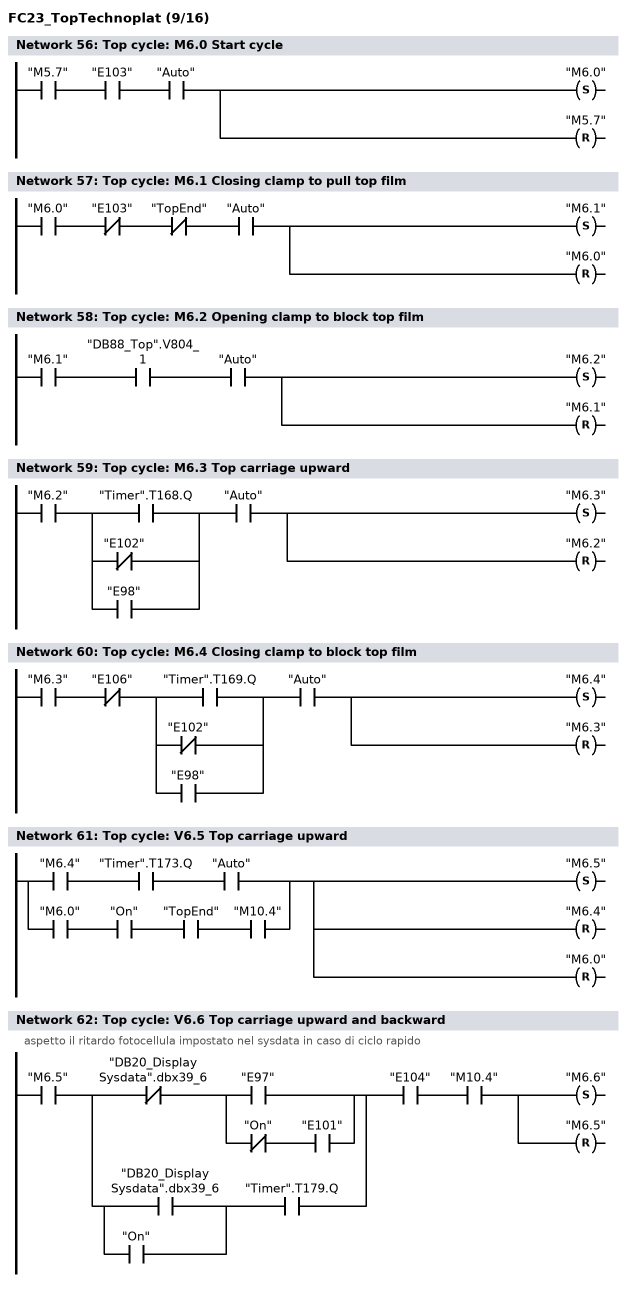
   RUNG wire#powerrail
      Contact( "M5.7" )
      Contact( "E103" )
      Contact( "Auto" )
      wire#w1
      S_Coil( "M6.0" )
   END_RUNG
   RUNG wire#w1
      R_Coil( "M5.7" )
   END_RUNG
   // the same network as SCL:
   IF "M5.7" AND "E103" AND "Auto" THEN
       "M6.0" := TRUE;
       "M5.7" := FALSE;
   END_IF;
END_REGION

REGION Network 57: Top cycle: M6.1 Closing clamp to pull top film
   RUNG wire#powerrail
      Contact( "M6.0" )
      I_Contact( "E103" )
      I_Contact( "TopEnd" )
      Contact( "Auto" )
      wire#w1
      S_Coil( "M6.1" )
   END_RUNG
   RUNG wire#w1
      R_Coil( "M6.0" )
   END_RUNG
   // the same network as SCL:
   IF "M6.0" AND NOT "E103" AND NOT "TopEnd" AND "Auto" THEN
       "M6.1" := TRUE;
       "M6.0" := FALSE;
   END_IF;
END_REGION

REGION Network 58: Top cycle: M6.2 Opening clamp to block top film
   RUNG wire#powerrail
      Contact( "M6.1" )
      Contact( "DB88_Top".V804_1 )
      Contact( "Auto" )
      wire#w1
      S_Coil( "M6.2" )
   END_RUNG
   RUNG wire#w1
      R_Coil( "M6.1" )
   END_RUNG
   // the same network as SCL:
   IF "M6.1" AND "DB88_Top".V804_1 AND "Auto" THEN
       "M6.2" := TRUE;
       "M6.1" := FALSE;
   END_IF;
END_REGION

REGION Network 59: Top cycle: M6.3 Top carriage upward
   RUNG wire#powerrail
      Contact( "M6.2" )
      wire#w1
      Contact( "Timer".T168.Q )
      wire#w2
      Contact( "Auto" )
      wire#w3
      S_Coil( "M6.3" )
   END_RUNG
   RUNG wire#w1
      I_Contact( "E102" )
   END_RUNG wire#w2
   RUNG wire#w1
      Contact( "E98" )
   END_RUNG wire#w2
   RUNG wire#w3
      R_Coil( "M6.2" )
   END_RUNG
   // the same network as SCL:
   IF "M6.2" AND ("Timer".T168.Q OR NOT "E102" OR "E98") AND "Auto" THEN
       "M6.3" := TRUE;
       "M6.2" := FALSE;
   END_IF;
END_REGION

REGION Network 60: Top cycle: M6.4 Closing clamp to block top film
   RUNG wire#powerrail
      Contact( "M6.3" )
      I_Contact( "E106" )
      wire#w1
      Contact( "Timer".T169.Q )
      wire#w2
      Contact( "Auto" )
      wire#w3
      S_Coil( "M6.4" )
   END_RUNG
   RUNG wire#w1
      I_Contact( "E102" )
   END_RUNG wire#w2
   RUNG wire#w1
      Contact( "E98" )
   END_RUNG wire#w2
   RUNG wire#w3
      R_Coil( "M6.3" )
   END_RUNG
   // the same network as SCL:
   IF "M6.3" AND NOT "E106" AND ("Timer".T169.Q OR NOT "E102" OR "E98") AND "Auto" THEN
       "M6.4" := TRUE;
       "M6.3" := FALSE;
   END_IF;
END_REGION

REGION Network 61: Top cycle: V6.5 Top carriage upward
   RUNG wire#powerrail
      Contact( "M6.4" )
      Contact( "Timer".T173.Q )
      Contact( "Auto" )
      wire#w1
      S_Coil( "M6.5" )
   END_RUNG
   RUNG wire#powerrail
      Contact( "M6.0" )
      Contact( "On" )
      Contact( "TopEnd" )
      Contact( "M10.4" )
   END_RUNG wire#w1
   RUNG wire#w1
      R_Coil( "M6.4" )
   END_RUNG
   RUNG wire#w1
      R_Coil( "M6.0" )
   END_RUNG
   // the same network as SCL:
   IF ("M6.4" AND "Timer".T173.Q AND "Auto") OR ("M6.0" AND "On" AND "TopEnd" AND "M10.4") THEN
       "M6.5" := TRUE;
   END_IF;
   #_w1 := ("M6.4" AND "Timer".T173.Q AND "Auto") OR ("M6.0" AND "On" AND "TopEnd" AND "M10.4");
   IF #_w1 THEN
       "M6.4" := FALSE;
       "M6.0" := FALSE;
   END_IF;
END_REGION

REGION Network 62: Top cycle: V6.6 Top carriage upward and backward
   // aspetto il ritardo fotocellula impostato nel sysdata in caso di ciclo rapido
   RUNG wire#powerrail
      Contact( "M6.5" )
      wire#w1
      I_Contact( "DB20_DisplaySysdata".dbx39_6 )
      wire#w2
      Contact( "E97" )
      wire#w3
      Contact( "E104" )
      Contact( "M10.4" )
      wire#w5
      S_Coil( "M6.6" )
   END_RUNG
   RUNG wire#w2
      I_Contact( "On" )
      Contact( "E101" )
   END_RUNG wire#w3
   RUNG wire#w1
      Contact( "DB20_DisplaySysdata".dbx39_6 )
      wire#w4
      Contact( "Timer".T179.Q )
   END_RUNG wire#w3
   RUNG wire#w1
      Contact( "On" )
   END_RUNG wire#w4
   RUNG wire#w5
      R_Coil( "M6.5" )
   END_RUNG
   // the same network as SCL:
   IF "M6.5" AND ((NOT "DB20_DisplaySysdata".dbx39_6 AND ("E97" OR (NOT "On" AND "E101"))) OR (("DB20_DisplaySysdata".dbx39_6 OR "On") AND "Timer".T179.Q)) AND "E104" AND "M10.4" THEN
       "M6.6" := TRUE;
       "M6.5" := FALSE;
   END_IF;
END_REGION

REGION Network 63: Top cycle: M6.7 Top cutter backward
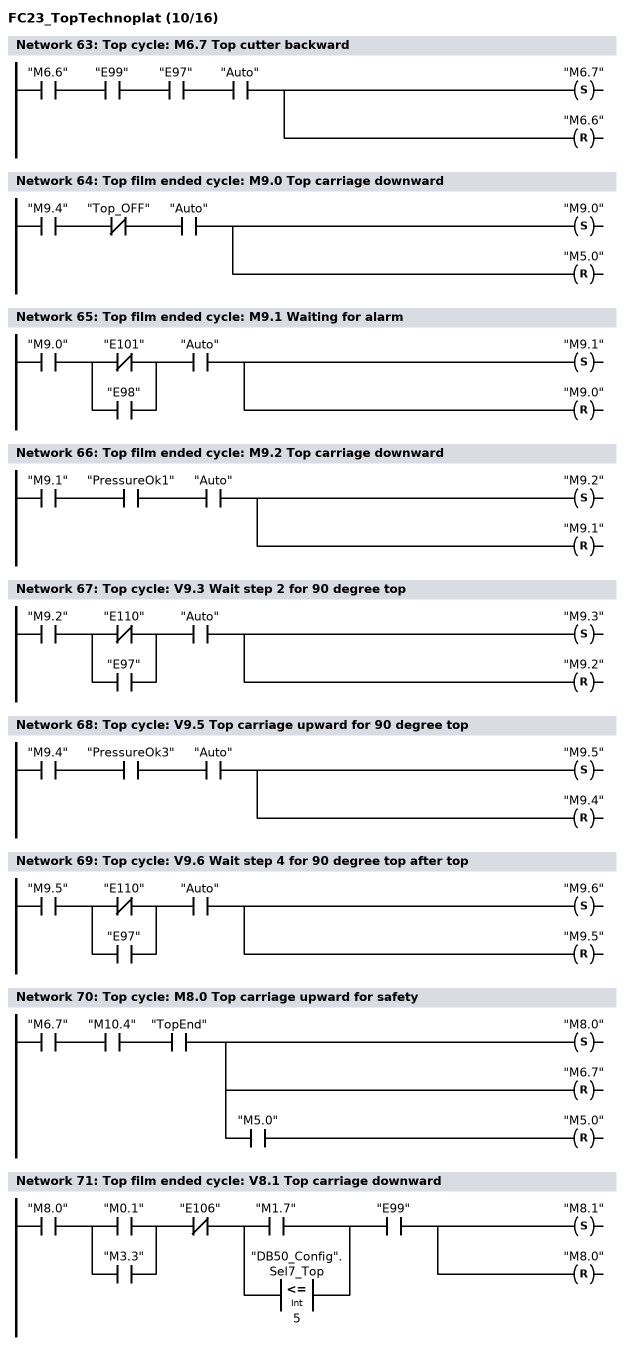
   RUNG wire#powerrail
      Contact( "M6.6" )
      Contact( "E99" )
      Contact( "E97" )
      Contact( "Auto" )
      wire#w1
      S_Coil( "M6.7" )
   END_RUNG
   RUNG wire#w1
      R_Coil( "M6.6" )
   END_RUNG
   // the same network as SCL:
   IF "M6.6" AND "E99" AND "E97" AND "Auto" THEN
       "M6.7" := TRUE;
       "M6.6" := FALSE;
   END_IF;
END_REGION

REGION Network 64: Top film ended cycle: M9.0 Top carriage downward
   RUNG wire#powerrail
      Contact( "M9.4" )
      I_Contact( "Top_OFF" )
      Contact( "Auto" )
      wire#w1
      S_Coil( "M9.0" )
   END_RUNG
   RUNG wire#w1
      R_Coil( "M5.0" )
   END_RUNG
   // the same network as SCL:
   IF "M9.4" AND NOT "Top_OFF" AND "Auto" THEN
       "M9.0" := TRUE;
       "M5.0" := FALSE;
   END_IF;
END_REGION

REGION Network 65: Top film ended cycle: M9.1 Waiting for alarm
   RUNG wire#powerrail
      Contact( "M9.0" )
      wire#w1
      I_Contact( "E101" )
      wire#w2
      Contact( "Auto" )
      wire#w3
      S_Coil( "M9.1" )
   END_RUNG
   RUNG wire#w1
      Contact( "E98" )
   END_RUNG wire#w2
   RUNG wire#w3
      R_Coil( "M9.0" )
   END_RUNG
   // the same network as SCL:
   IF "M9.0" AND (NOT "E101" OR "E98") AND "Auto" THEN
       "M9.1" := TRUE;
       "M9.0" := FALSE;
   END_IF;
END_REGION

REGION Network 66: Top film ended cycle: M9.2 Top carriage downward
   RUNG wire#powerrail
      Contact( "M9.1" )
      Contact( "PressureOk1" )
      Contact( "Auto" )
      wire#w1
      S_Coil( "M9.2" )
   END_RUNG
   RUNG wire#w1
      R_Coil( "M9.1" )
   END_RUNG
   // the same network as SCL:
   IF "M9.1" AND "PressureOk1" AND "Auto" THEN
       "M9.2" := TRUE;
       "M9.1" := FALSE;
   END_IF;
END_REGION

REGION Network 67: Top cycle: V9.3 Wait step 2 for 90 degree top
   RUNG wire#powerrail
      Contact( "M9.2" )
      wire#w1
      I_Contact( "E110" )
      wire#w2
      Contact( "Auto" )
      wire#w3
      S_Coil( "M9.3" )
   END_RUNG
   RUNG wire#w1
      Contact( "E97" )
   END_RUNG wire#w2
   RUNG wire#w3
      R_Coil( "M9.2" )
   END_RUNG
   // the same network as SCL:
   IF "M9.2" AND (NOT "E110" OR "E97") AND "Auto" THEN
       "M9.3" := TRUE;
       "M9.2" := FALSE;
   END_IF;
END_REGION

REGION Network 68: Top cycle: V9.5 Top carriage upward for 90 degree top
   RUNG wire#powerrail
      Contact( "M9.4" )
      Contact( "PressureOk3" )
      Contact( "Auto" )
      wire#w1
      S_Coil( "M9.5" )
   END_RUNG
   RUNG wire#w1
      R_Coil( "M9.4" )
   END_RUNG
   // the same network as SCL:
   IF "M9.4" AND "PressureOk3" AND "Auto" THEN
       "M9.5" := TRUE;
       "M9.4" := FALSE;
   END_IF;
END_REGION

REGION Network 69: Top cycle: V9.6 Wait step 4 for 90 degree top after top
   RUNG wire#powerrail
      Contact( "M9.5" )
      wire#w1
      I_Contact( "E110" )
      wire#w2
      Contact( "Auto" )
      wire#w3
      S_Coil( "M9.6" )
   END_RUNG
   RUNG wire#w1
      Contact( "E97" )
   END_RUNG wire#w2
   RUNG wire#w3
      R_Coil( "M9.5" )
   END_RUNG
   // the same network as SCL:
   IF "M9.5" AND (NOT "E110" OR "E97") AND "Auto" THEN
       "M9.6" := TRUE;
       "M9.5" := FALSE;
   END_IF;
END_REGION

REGION Network 70: Top cycle: M8.0 Top carriage upward for safety
   RUNG wire#powerrail
      Contact( "M6.7" )
      Contact( "M10.4" )
      Contact( "TopEnd" )
      wire#w1
      S_Coil( "M8.0" )
   END_RUNG
   RUNG wire#w1
      R_Coil( "M6.7" )
   END_RUNG
   RUNG wire#w1
      Contact( "M5.0" )
      R_Coil( "M5.0" )
   END_RUNG
   // the same network as SCL:
   #_w1 := "M6.7" AND "M10.4" AND "TopEnd";
   IF #_w1 THEN
       "M8.0" := TRUE;
       "M6.7" := FALSE;
   END_IF;
   IF #_w1 AND "M5.0" THEN "M5.0" := FALSE; END_IF;
END_REGION

REGION Network 71: Top film ended cycle: V8.1 Top carriage downward
   RUNG wire#powerrail
      Contact( "M8.0" )
      wire#w1
      Contact( "M0.1" )
      wire#w2
      I_Contact( "E106" )
      wire#w3
      Contact( "M1.7" )
      wire#w4
      Contact( "E99" )
      wire#w5
      S_Coil( "M8.1" )
   END_RUNG
   RUNG wire#w1
      Contact( "M3.3" )
   END_RUNG wire#w2
   RUNG wire#w3
      { S7_Templates := "SrcType := Int" } LE_Contact(in1 := "DB50_Config".Sel7_Top, in2 := 5)
   END_RUNG wire#w4
   RUNG wire#w5
      R_Coil( "M8.0" )
   END_RUNG
   // the same network as SCL:
   IF "M8.0" AND ("M0.1" OR "M3.3") AND NOT "E106" AND ("M1.7" OR ("DB50_Config".Sel7_Top <= 5)) AND "E99" THEN
       "M8.1" := TRUE;
       "M8.0" := FALSE;
   END_IF;
END_REGION

REGION Network 72: Top film ended cycle: V8.2 Top carriage forward
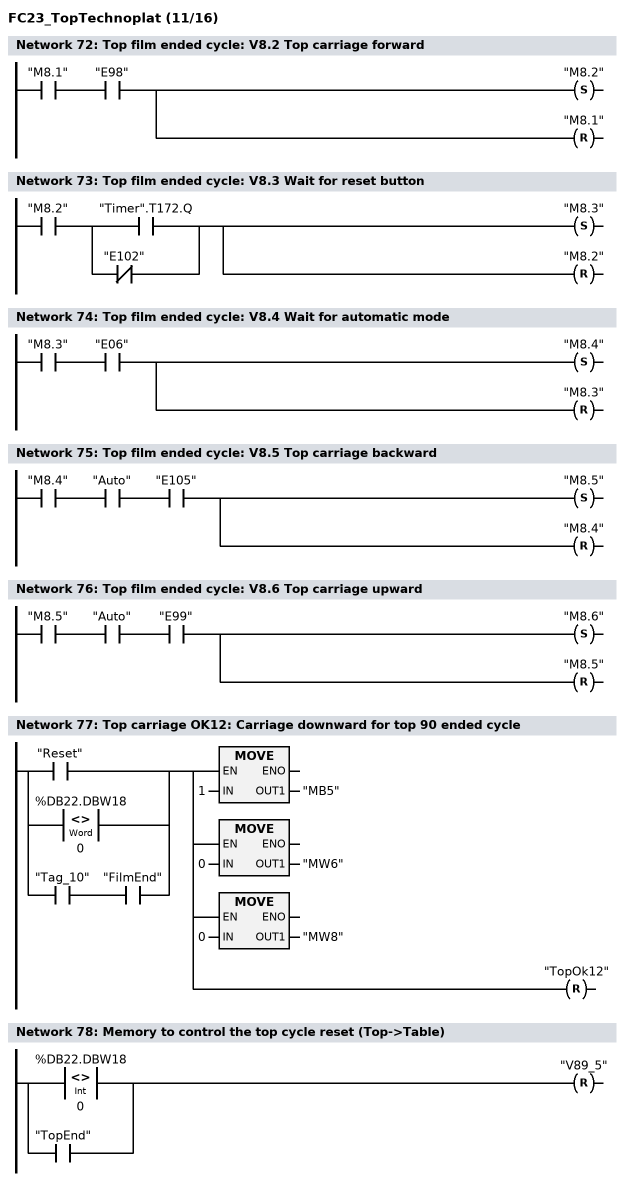
   RUNG wire#powerrail
      Contact( "M8.1" )
      Contact( "E98" )
      wire#w1
      S_Coil( "M8.2" )
   END_RUNG
   RUNG wire#w1
      R_Coil( "M8.1" )
   END_RUNG
   // the same network as SCL:
   IF "M8.1" AND "E98" THEN
       "M8.2" := TRUE;
       "M8.1" := FALSE;
   END_IF;
END_REGION

REGION Network 73: Top film ended cycle: V8.3 Wait for reset button
   RUNG wire#powerrail
      Contact( "M8.2" )
      wire#w1
      Contact( "Timer".T172.Q )
      wire#w2
      S_Coil( "M8.3" )
   END_RUNG
   RUNG wire#w1
      I_Contact( "E102" )
   END_RUNG wire#w2
   RUNG wire#w2
      R_Coil( "M8.2" )
   END_RUNG
   // the same network as SCL:
   IF "M8.2" AND ("Timer".T172.Q OR NOT "E102") THEN
       "M8.3" := TRUE;
       "M8.2" := FALSE;
   END_IF;
END_REGION

REGION Network 74: Top film ended cycle: V8.4 Wait for automatic mode
   RUNG wire#powerrail
      Contact( "M8.3" )
      Contact( "E06" )
      wire#w1
      S_Coil( "M8.4" )
   END_RUNG
   RUNG wire#w1
      R_Coil( "M8.3" )
   END_RUNG
   // the same network as SCL:
   IF "M8.3" AND "E06" THEN
       "M8.4" := TRUE;
       "M8.3" := FALSE;
   END_IF;
END_REGION

REGION Network 75: Top film ended cycle: V8.5 Top carriage backward
   RUNG wire#powerrail
      Contact( "M8.4" )
      Contact( "Auto" )
      Contact( "E105" )
      wire#w1
      S_Coil( "M8.5" )
   END_RUNG
   RUNG wire#w1
      R_Coil( "M8.4" )
   END_RUNG
   // the same network as SCL:
   IF "M8.4" AND "Auto" AND "E105" THEN
       "M8.5" := TRUE;
       "M8.4" := FALSE;
   END_IF;
END_REGION

REGION Network 76: Top film ended cycle: V8.6 Top carriage upward
   RUNG wire#powerrail
      Contact( "M8.5" )
      Contact( "Auto" )
      Contact( "E99" )
      wire#w1
      S_Coil( "M8.6" )
   END_RUNG
   RUNG wire#w1
      R_Coil( "M8.5" )
   END_RUNG
   // the same network as SCL:
   IF "M8.5" AND "Auto" AND "E99" THEN
       "M8.6" := TRUE;
       "M8.5" := FALSE;
   END_IF;
END_REGION

REGION Network 77: Top carriage OK12: Carriage downward for top 90 ended cycle
   RUNG wire#powerrail
      Contact( "Reset" )
      wire#w1
      { S7_GenerateENO := "TRUE" } Move(in := 1, out1 => "MB5")
   END_RUNG
   RUNG wire#powerrail
      { S7_Templates := "SrcType := Word" } NE_Contact(in1 := %DB22.DBW18, in2 := 0)
   END_RUNG wire#w1
   RUNG wire#powerrail
      Contact( "Tag_10" )
      Contact( "FilmEnd" )
   END_RUNG wire#w1
   RUNG wire#w1
      { S7_GenerateENO := "TRUE" } Move(in := 0, out1 => "MW6")
   END_RUNG
   RUNG wire#w1
      { S7_GenerateENO := "TRUE" } Move(in := 0, out1 => "MW8")
   END_RUNG
   RUNG wire#w1
      R_Coil( "TopOk12" )
   END_RUNG
   // the same network as SCL:
   IF "Reset" OR (%DB22.DBW18 <> 0) OR ("Tag_10" AND "FilmEnd") THEN
       "MB5" := 1;
       "MW6" := 0;
       "MW8" := 0;
       "TopOk12" := FALSE;
   END_IF;
END_REGION

REGION Network 78: Memory to control the top cycle reset (Top->Table)
   RUNG wire#powerrail
      { S7_Templates := "SrcType := Int" } NE_Contact(in1 := %DB22.DBW18, in2 := 0)
      wire#w1
      R_Coil( "V89_5" )
   END_RUNG
   RUNG wire#powerrail
      Contact( "TopEnd" )
   END_RUNG wire#w1
   // the same network as SCL:
   IF (%DB22.DBW18 <> 0) OR "TopEnd" THEN "V89_5" := FALSE; END_IF;
END_REGION

REGION Network 79: Top carriage forward (Top)
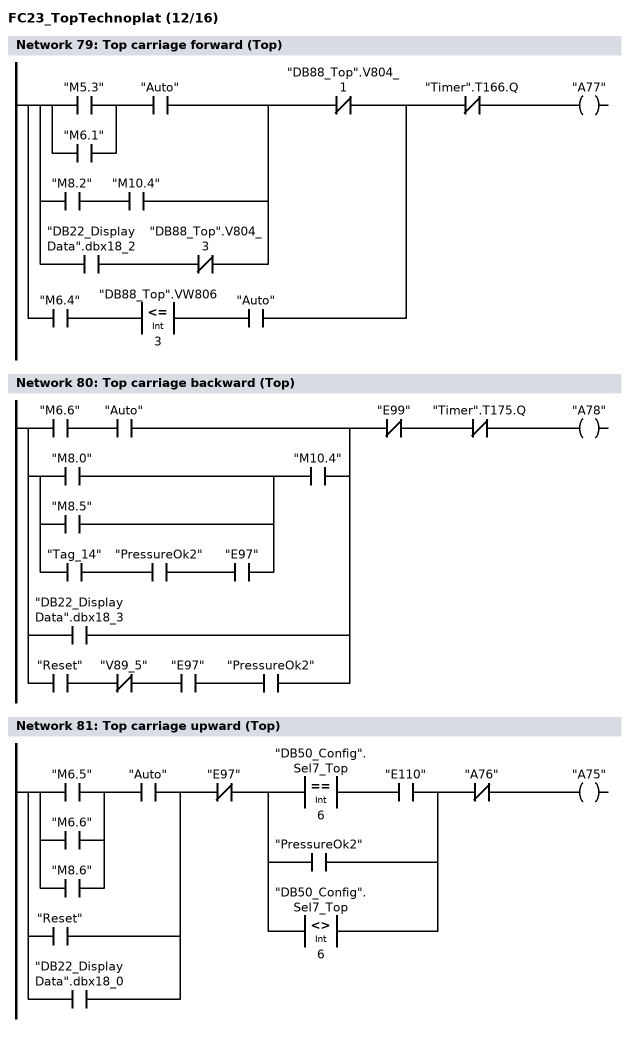
   RUNG wire#powerrail
      Contact( "M5.3" )
      wire#w1
      Contact( "Auto" )
      wire#w2
      I_Contact( "DB88_Top".V804_1 )
      wire#w3
      I_Contact( "Timer".T166.Q )
      Coil( "A77" )
   END_RUNG
   RUNG wire#powerrail
      Contact( "M6.1" )
   END_RUNG wire#w1
   RUNG wire#powerrail
      Contact( "M8.2" )
      Contact( "M10.4" )
   END_RUNG wire#w2
   RUNG wire#powerrail
      Contact( "DB22_DisplayData".dbx18_2 )
      I_Contact( "DB88_Top".V804_3 )
   END_RUNG wire#w2
   RUNG wire#powerrail
      Contact( "M6.4" )
      { S7_Templates := "SrcType := Int" } LE_Contact(in1 := "DB88_Top".VW806, in2 := 3)
      Contact( "Auto" )
   END_RUNG wire#w3
   // the same network as SCL:
   "A77" := ((((("M5.3" OR "M6.1") AND "Auto") OR ("M8.2" AND "M10.4") OR ("DB22_DisplayData".dbx18_2 AND NOT "DB88_Top".V804_3)) AND NOT "DB88_Top".V804_1) OR ("M6.4" AND ("DB88_Top".VW806 <= 3) AND "Auto")) AND NOT "Timer".T166.Q;
END_REGION

REGION Network 80: Top carriage backward (Top)
   RUNG wire#powerrail
      Contact( "M6.6" )
      Contact( "Auto" )
      wire#w1
      I_Contact( "E99" )
      I_Contact( "Timer".T175.Q )
      Coil( "A78" )
   END_RUNG
   RUNG wire#powerrail
      Contact( "M8.0" )
      wire#w2
      Contact( "M10.4" )
   END_RUNG wire#w1
   RUNG wire#powerrail
      Contact( "M8.5" )
   END_RUNG wire#w2
   RUNG wire#powerrail
      Contact( "Tag_14" )
      Contact( "PressureOk2" )
      Contact( "E97" )
   END_RUNG wire#w2
   RUNG wire#powerrail
      Contact( "DB22_DisplayData".dbx18_3 )
   END_RUNG wire#w1
   RUNG wire#powerrail
      Contact( "Reset" )
      I_Contact( "V89_5" )
      Contact( "E97" )
      Contact( "PressureOk2" )
   END_RUNG wire#w1
   // the same network as SCL:
   "A78" := (("M6.6" AND "Auto") OR (("M8.0" OR "M8.5" OR ("Tag_14" AND "PressureOk2" AND "E97")) AND "M10.4") OR "DB22_DisplayData".dbx18_3 OR ("Reset" AND NOT "V89_5" AND "E97" AND "PressureOk2")) AND NOT "E99" AND NOT "Timer".T175.Q;
END_REGION

REGION Network 81: Top carriage upward (Top)
   RUNG wire#powerrail
      Contact( "M6.5" )
      wire#w1
      Contact( "Auto" )
      wire#w2
      I_Contact( "E97" )
      wire#w3
      { S7_Templates := "SrcType := Int" } EQ_Contact(in1 := "DB50_Config".Sel7_Top, in2 := 6)
      Contact( "E110" )
      wire#w4
      I_Contact( "A76" )
      Coil( "A75" )
   END_RUNG
   RUNG wire#powerrail
      Contact( "M6.6" )
   END_RUNG wire#w1
   RUNG wire#powerrail
      Contact( "M8.6" )
   END_RUNG wire#w1
   RUNG wire#powerrail
      Contact( "Reset" )
   END_RUNG wire#w2
   RUNG wire#powerrail
      Contact( "DB22_DisplayData".dbx18_0 )
   END_RUNG wire#w2
   RUNG wire#w3
      Contact( "PressureOk2" )
   END_RUNG wire#w4
   RUNG wire#w3
      { S7_Templates := "SrcType := Int" } NE_Contact(in1 := "DB50_Config".Sel7_Top, in2 := 6)
   END_RUNG wire#w4
   // the same network as SCL:
   "A75" := ((("M6.5" OR "M6.6" OR "M8.6") AND "Auto") OR "Reset" OR "DB22_DisplayData".dbx18_0) AND NOT "E97" AND ((("DB50_Config".Sel7_Top = 6) AND "E110") OR "PressureOk2" OR ("DB50_Config".Sel7_Top <> 6)) AND NOT "A76";
END_REGION

REGION Network 82: Top carriage downward (Top)
